(* IEC 61131-3 sources: brOscatLib/oscatNetw, 129 files *)

(* ---- oscatNetw.typ ---- *)
TYPE
    DLOG_CRON_DATA :    STRUCT
        CE : ARRAY[0..5] OF DLOG_CRON_ELEMENT;
    END_STRUCT;
    DLOG_CRON_ELEMENT :    STRUCT
        ELEMENTS : ARRAY[0..59] OF BOOL;
        VALUE : INT;
        VALUE_MIN : INT;
        VALUE_MAX : INT;
        ALL_SELECTED : BOOL;
    END_STRUCT;
    DLOG_DATA :    STRUCT
        STORE_TYPE : BYTE;
        ADD_COM : INT;
        ADD_DATA_REQ : BOOL;
        CLOCK_TRIG : BOOL;
        ID_MAX : USINT;
        DTI : DT;
        UCB : UNI_CIRCULAR_BUFFER_DATA;
        LOAD_TIME_MAX : TIME;
        NEW_FILE : STRING[255];
        NEW_FILE_SIZE : UDINT;
        NEW_FILE_RTRIG : BOOL;
    END_STRUCT;
    DLOG_REAL_ARRAY_ELEMENT :    STRUCT
        VALUE : REAL;
        DELTA : REAL;
        COLUMN : STRING[10];
        _DELTA_LAST : REAL;
        _VALUE_LAST : REAL;
    END_STRUCT;
    DLOG_RETAIN :    STRUCT
        FN_REM : STRING[255];
        COLOR : BOOL;
        HEAD : BOOL;
        TRIG_CNT : UDINT;
        TRIG_CNT_TOTAL : UDINT;
    END_STRUCT;
    DLOG_SAVE :    STRUCT
        FN_REM : STRING[255];
        COLOR : BOOL;
        HEAD : BOOL;
        TRIG_CNT : UDINT;
        TRIG_CNT_TOTAL : UDINT;
    END_STRUCT;
    LOG_CONTROL :    STRUCT
        NEW_MSG : STRING[LOG_SIZE]; (* neue Nachricht für den Datenbuffer *)
        NEW_MSG_OPTION : DWORD;
        LEVEL : BYTE;
        SIZE : INT := LOG_MAX; (* Anzahl der Strings im LOG_DATA *)
        RESET : BOOL; (* Nachrichtenbuffer löschen *)
        PRINTF : PRINTF_DATA; (* Array PRINTF Parameter *)
        MSG : ARRAY[0..LOG_MAX] OF STRING[LOG_SIZE]; (* Array Message *)
        MSG_OPTION : ARRAY[0..LOG_MAX] OF DWORD; (* Array Options *)
        UPDATE_COUNT : UINT; (* Updatezähler *)
        IDX : INT; (* aktueller Nachrichten-Index *)
        RING_MODE : BOOL; (* Bufferüberlauf erkannt *)
    END_STRUCT;
    UNI_CIRCULAR_BUFFER_DATA :    STRUCT
        D_MODE : INT;
        D_SIZE : INT;
        D_HEAD : WORD;
        D_STRING : STRING[STRING_LENGTH];
        D_REAL : REAL;
        D_DWORD : DWORD;
        BUF_SIZE : UINT;
        BUF_COUNT : UINT;
        BUF_USED : USINT;
        BUF_USED_MAX : USINT;
        BUF_DATA_CNT : UDINT;
        BUF_DATA_LOST : UDINT;
        BUF : UNI_CIRCULAR_BUF;
        _GetStart : UINT;
        _GetEnd : UINT;
        _Last : UINT;
        _First : UINT;
    END_STRUCT;
    us_LOG_VIEWPORT :    STRUCT
        LINE_ARRAY : ARRAY[1..40] OF INT;
        COUNT : INT; (* Anzahl der sichtbaren Nachtrichten *)
        UPDATE_COUNT : UINT; (* Updatezähler *)
        MOVE_TO_X : INT; (* Steuerung der Nachrichtenanzeige *)
        UPDATE : BOOL; (* Daten wurden geändert -> neuzeichnen *)
    END_STRUCT;
    MYSQL_COM :    STRUCT
        S_BUF : NETWORK_BUFFER;
        R_BUF : NETWORK_BUFFER;
        SQL_CON : BOOL;
        SQL_URL : STRING[STRING_LENGTH];
        SQL_PACKET_NO : BYTE;
        TIMEOUT : TIME;
        DNS_IP4 : DWORD;
        SQL_RCV_STATE : BYTE;
        ERROR_C : DWORD;
        ERROR_T : BYTE;
    END_STRUCT;
    MYSQL_INFO :    STRUCT
        SERVER_PROTOCOL_VERSION : BYTE;
        SERVER_CAPABILITIES : WORD;
        SERVER_STATUS : WORD;
        SERVER_LANGUAGE : BYTE;
        SQL_CONNECTED : BOOL;
        SQL_ERROR : STRING[STRING_LENGTH];
        DATA_INSERT_AKTIV : BOOL;
        DATA_INSERT_OK_CNT : UDINT;
        DATA_INSERT_NOK_CNT : UDINT;
    END_STRUCT;
    FILE_PATH_DATA :    STRUCT
        DRIVE : STRING[3];
        DIRECTORY : STRING[STRING_LENGTH];
        FILENAME : STRING[255];
    END_STRUCT;
    FILE_SERVER_DATA :    STRUCT
        FILE_OPEN : BOOL;
        FILENAME : STRING[255];
        MODE : BYTE;
        OFFSET : UDINT;
        FILE_SIZE : UDINT;
        ERROR : BYTE;
        RUNTIME : FILE_SERVER_RUNTIME_DATA;
    END_STRUCT;
    FILE_SERVER_RUNTIME_DATA :    STRUCT
        TIME_FILE_OPEN_CUR : UDINT;
        TIME_FILE_OPEN_MAX : UDINT;
        TIME_FILE_OPEN_MIN : UDINT;
        TIME_FILE_CLOSE_CUR : UDINT;
        TIME_FILE_CLOSE_MAX : UDINT;
        TIME_FILE_CLOSE_MIN : UDINT;
        TIME_FILE_READ_CUR : UDINT;
        TIME_FILE_READ_MAX : UDINT;
        TIME_FILE_READ_MIN : UDINT;
        TIME_FILE_WRITE_CUR : UDINT;
        TIME_FILE_WRITE_MAX : UDINT;
        TIME_FILE_WRITE_MIN : UDINT;
        TIME_FILE_SEEK_CUR : UDINT;
        TIME_FILE_SEEK_MAX : UDINT;
        TIME_FILE_SEEK_MIN : UDINT;
        TIME_FILE_TELL_CUR : UDINT;
        TIME_FILE_TELL_MAX : UDINT;
        TIME_FILE_TELL_MIN : UDINT;
        TIME_FILE_DELETE_CUR : UDINT;
        TIME_FILE_DELETE_MAX : UDINT;
        TIME_FILE_DELETE_MIN : UDINT;
    END_STRUCT;
    NET_VAR_DATA :    STRUCT
        CYCLE : UDINT;
        STATE : BYTE;
        INDEX : INT;
        ID_MAX : USINT;
        ERROR_ID : BYTE;
        BUF_SIZE : UINT;
        S_BUF : NETWORK_BUFFER;
        R_BUF : NETWORK_BUFFER;
    END_STRUCT;
    IP2GEO_DATA :    STRUCT
        STATE : BOOL;
        IP4 : DWORD;
        COUNTRY_CODE : STRING[2];
        COUNTRY_NAME : STRING[20];
        REGION_CODE : STRING[2];
        REGION_NAME : STRING[20];
        CITY : STRING[20];
        GEO_LATITUDE : REAL;
        GEO_LONGITUDE : REAL;
        TIME_ZONE_NAME : STRING[20];
        GMT_OFFSET : INT;
        IS_DST : BOOL;
    END_STRUCT;
    IP_C :    STRUCT
        C_MODE : BYTE; (*W Mode: TCP/UCP AKTIV/PASSIV                               *)
        C_PORT : WORD; (*W Portnummer                                               *)
        C_IP : DWORD; (*W IP-Adresse gepackt wwxxyyzz = www.xxx.yyy.zzz            *)
        C_STATE : BYTE; (*R Verbindungsstatus ON/OFF + Flanke ON/OFF                 *)
        C_ENABLE : BOOL; (*W Freigabe für Connect                                     *)
        R_OBSERVE : BOOL; (*W Empfang ueberwachen                                      *)
        TIME_RESET : BOOL; (*W Alle Timer ruecksetzen                                   *)
        ERROR : DWORD; (*R vvwwxxyy (vv = CON_ERROR, ww = SEN_ERROR, xx = REC_ERROR *)
        FIFO : IP_FIFO_DATA; (*I IP FIFO Struktur                                         *)
        MAILBOX : ARRAY[1..16] OF BYTE; (*I Mailbox: Datenbereich für Bausteindatenaustausch         *)
    END_STRUCT;
    IP_FIFO_DATA :    STRUCT
        X : ARRAY[1..128] OF BYTE; (* IP_ID FIFO Speicher          *)
        Y : ARRAY[1..128] OF BYTE; (* IP_ID Zähler                 *)
        ID : BYTE; (* höchste vergabene id         *)
        MAX_ID : BYTE; (* maximal Anmeldungen pro ID   *)
        INIT : BOOL; (* Initialisierung durchgeführt *)
        EMPTY : BOOL; (* FIFO leer                    *)
        FULL : BOOL; (* FIFO voll                    *)
        TOP : INT; (* maximale anzahl in FIFO      *)
        NW : INT; (* Schreibzeiger                *)
        NR : INT; (* Lesezeiger                   *)
    END_STRUCT;
    NETWORK_BUFFER :    STRUCT
        SIZE : UINT;
        BUFFER : NW_BUF_LONG;
    END_STRUCT;
    NETWORK_BUFFER_SHORT :    STRUCT
        SIZE : UINT;
        BUFFER : NW_BUF_SHORT;
    END_STRUCT;
    URL :    STRUCT
        PROTOCOL : STRING[10];
        USER : STRING[32];
        PASSWORD : STRING[32];
        DOMAIN : STRING[80];
        PORT : WORD;
        PATH : STRING[80];
        QUERY : STRING[STRING_LENGTH];
        ANCHOR : STRING[40];
        HEADER : STRING[160];
    END_STRUCT;
    VMAP_DATA :    STRUCT
        FC : DWORD;
        V_ADR : INT;
        V_SIZE : INT;
        P_ADR : INT;
        TIME_OUT : TIME;
    END_STRUCT;
    XML_CONTROL :    STRUCT
        COMMAND : WORD;
        WATCHDOG : TIME;
        START_POS : UINT;
        STOP_POS : UINT;
        COUNT : UINT;
        TYP : INT;
        LEVEL : UINT;
        PATH : STRING[STRING_LENGTH];
        ELEMENT : STRING[STRING_LENGTH];
        ATTRIBUTE : STRING[STRING_LENGTH];
        VALUE : STRING[STRING_LENGTH];
        BLOCK1_START : UINT;
        BLOCK1_STOP : UINT;
        BLOCK2_START : UINT;
        BLOCK2_STOP : UINT;
    END_STRUCT;
    us_TN_INPUT_CONTROL :    STRUCT
        bo_Enable : BOOL; (* Bearbeitung freigeben/sperren *)
        bo_Update_all : BOOL; (* All Elemente neu zeichnen *)
        bo_Reset_Fokus : BOOL; (* Fokus auf 1. Element setzen *)
        in_Focus_at : INT; (* Controlelement mit aktivem Fokus *)
        in_Count : INT; (* Anzahl der benutzen Control-Elemente *)
        in_ToolTip_X : INT; (* Tooltip Text X-Offset *)
        in_ToolTip_Y : INT; (* Tooltip Text Y-Offset *)
        by_ToolTip_Attr : BYTE; (* Tooltip Text Attribute *)
        in_ToolTip_Size : INT; (* Tooltip Text länge *)
        usa_TN_INPUT_CONTROL_DATA : ARRAY[1..20] OF us_TN_INPUT_CONTROL_DATA;
    END_STRUCT;
    us_TN_INPUT_CONTROL_DATA :    STRUCT
        by_Input_Exten_Code : BYTE;
        by_Input_ASCII_Code : BYTE;
        bo_Input_ASCII_IsNum : BOOL;
        in_Title_X_Offset : INT; (* Title Text X-Offset *)
        in_Title_Y_Offset : INT; (* Title Text Y-Offset *)
        by_Title_Attr : BYTE; (* Title Text Attribute *)
        st_Title_String : STRING[255]; (* Title Text String *)
        in_Cursor_X : INT; (* aktuelle Cursor X-Position *)
        in_Cursor_Y : INT; (* aktuelle Cursor Y-Position *)
        in_Type : INT; (* Type des Elements *)
        in_X : INT; (* Element X-Position *)
        in_Y : INT; (* Element Y-Position *)
        in_Cursor_Pos : INT; (* aktuelle Cursorposition *)
        by_Attr_mF : BYTE; (* Text Attribute mit Fokus *)
        by_Attr_oF : BYTE; (* Text Attribute ohne Fokus *)
        in_selected : INT; (* Text Item wurde ausgewählt *)
        st_Input_Mask : STRING[255]; (* Text Eingabemaske *)
        st_Input_Data : STRING[STRING_LENGTH]; (* Text aktuelle Eingabedaten *)
        st_Input_String : STRING[255]; (* Text Kopie nach Return-Taste *)
        st_Input_ToolTip : STRING[255]; (* Text ToolTip (Eingabeinformation) *)
        in_Input_Option : INT; (* Text Ausgabe-Optionen *)
        bo_Input_Entered : BOOL; (* RETURN-Taste wurde betätigt *)
        bo_Input_Hidden : BOOL; (* Text versteckete Eingabe mit '*' *)
        bo_Input_Only_Num : BOOL; (* Text nur Nummerneingabe zulassen *)
        bo_Focus : BOOL; (* Element besitzt den Fokus *)
        bo_Update_Input : BOOL; (* Element wegen Benutzereingabe neuzeichnen *)
        bo_Update_All : BOOL; (* Element komplett neuzeichnen *)
    END_STRUCT;
    us_TN_MENU :    STRUCT
        st_Menu_Text : STRING[STRING_LENGTH]; (* X Menue Texte *)
        in_Menu_E_Count : INT; (* Menue Elemente Anzahl *)
        in_Y : INT; (* Menue Zeilennummer  Y-Position *)
        in_X : INT; (* Menue Spaltennummer X-Position *)
        by_Attr_mF : BYTE; (* Text Attribute mit Fokus *)
        by_Attr_oF : BYTE; (* Text Attribute ohne Fokus *)
        in_X_SM_new : INT; (* neue Sub-Menu X-Position *)
        in_Y_SM_new : INT; (* neue Sub-Menu Y-Position *)
        in_X_SM_old : INT; (* alte Sub-Menu X-Position *)
        in_Y_SM_old : INT; (* alte Sub-Menu Y-Position *)
        in_Cur_Menu_Item : INT; (* aktuelles Haupt-Menue *)
        in_Cur_Sub_Item : INT; (* aktuelles Sub-Menue *)
        in_State : INT; (*   Menu status   *)
        in_Menu_Selected : INT; (* X Menu-Item mit Enter angewwählt *)
        bo_Create : BOOL; (* X Menu erzeugen *)
        bo_Destroy : BOOL; (* X Menu entfernen *)
        bo_Update : BOOL; (* X Menu updaten *)
    END_STRUCT;
    us_TN_MENU_POPUP :    STRUCT
        st_Menu_Text : STRING[STRING_LENGTH]; (* X Menue Texte *)
        in_Menu_E_Count : INT; (* Menue Elemente Anzahl *)
        in_X : INT; (* X Menue X-Position *)
        in_Y : INT; (* X Menue Y-Position *)
        in_Cols : INT; (* Menue Spaltenanzahl *)
        in_Rows : INT; (* Menue Zeilenanzahl *)
        in_Cur_Item : INT; (* X aktuelles Sub-Menue *)
        by_Attr_mF : BYTE; (* X Text Attribute mit Fokus	*)
        by_Attr_oF : BYTE; (* X Text Attribute ohne Fokus *)
        by_Input_Exten_Code : BYTE; (* X Tastencode: Sondertasten *)
        bo_Create : BOOL; (* X Popup-Menu erzeugen *)
        bo_Destroy : BOOL; (* X Popup-Menu entfernen *)
        bo_Update : BOOL; (* X Popup-Menu updaten *)
        bo_Activ : BOOL; (*   Popup-Menu ist aktiv *)
    END_STRUCT;
    us_TN_SCREEN :    STRUCT
        bya_CHAR : ARRAY[0..1919] OF BYTE;
        bya_COLOR : ARRAY[0..1919] OF BYTE;
        bya_BACKUP : ARRAY[0..1919] OF BYTE;
        bya_Line_Update : ARRAY[0..23] OF BOOL;
        by_Input_Exten_Code : BYTE;
        by_Input_ASCII_Code : BYTE;
        bo_Input_ASCII_IsNum : BOOL;
        in_Page_Number : INT; (* aktive Seiten-Nr. *)
        in_Cursor_X : INT; (* Cursor X-Position *)
        in_Cursor_Y : INT; (* Cursor Y-Position *)
        in_EOS_Offset : INT; (* End of String Offset *)
        by_Clear_Screen_Attr : BYTE; (* Clear-Screen Attr *)
        bo_Clear_Screen : BOOL; (* Clear-Screen auslösen *)
        bo_Modal_Dialog : BOOL; (* Modaler Dialog ist aktiv *)
        bo_Menue_Bar_Dialog : BOOL; (* Menue Dialog ist aktiv *)
    END_STRUCT;
    WORLD_WEATHER_CUR :    STRUCT
        OBSERVATION_TIME : STRING[8];
        TEMP_C : INT;
        WEATHER_CODE : INT;
        WEATHER_DESC : STRING[60];
        WEATHER_ICON : INT;
        WIND_SPEED_MILES : INT;
        WIND_SPEED_KMPH : INT;
        WIND_DIR_DEGREE : INT;
        WIND_DIR16POINT : STRING[3];
        PRECIPMM : REAL;
        HUMIDITY : INT;
        VISIBILITY : INT;
        PRESSURE : INT;
        CLOUDOVER : INT;
    END_STRUCT;
    WORLD_WEATHER_DATA :    STRUCT
        CUR : WORLD_WEATHER_CUR;
        DAY : ARRAY[0..4] OF WORLD_WEATHER_DAY;
    END_STRUCT;
    WORLD_WEATHER_DAY :    STRUCT
        DATE_OF_DAY : STRING[10];
        TEMP_MAX_C : INT;
        TEMP_MAX_F : INT;
        TEMP_MIN_C : INT;
        TEMP_MIN_F : INT;
        WIND_SPEED_MILES : INT;
        WIND_SPEED_KMPH : INT;
        WIND_DIR_DEGREE : INT;
        WIND_DIR16POINT : STRING[3];
        WEATHER_CODE : INT;
        WEATHER_DESC : STRING[60];
        WEATHER_ICON : INT;
        PRECIPMM : REAL;
    END_STRUCT;
    YAHOO_WEATHER_DATA :    STRUCT
        LOCATION_CITY : STRING[40]; (* THE LOCATION OF THIS FORECAST: CITY: CITY NAME  *)
        LOCATION_REGION : STRING[20]; (* THE LOCATION OF THIS FORECAST: REGION: STATE, TERRITORY, OR REGION, IF GIVEN *)
        LOCATION_COUNTRY : STRING[20]; (* THE LOCATION OF THIS FORECAST: COUNTRY: TWO-CHARACTER COUNTRY CODE *)
        UNIT_TEMPERATURE : STRING[1]; (* TEMPERATURE: DEGREE UNITS, F FOR FAHRENHEIT OR C FOR CELSIUS *)
        UNIT_DISTANCE : STRING[2]; (* DISTANCE: UNITS FOR DISTANCE, MI FOR MILES OR KM FOR KILOMETERS *)
        UNIT_PRESSURE : STRING[2]; (* PRESSURE: UNITS OF BAROMETRIC PRESSURE, IN FOR POUNDS PER SQUARE INCH OR MB FOR MILLIBARS *)
        UNIT_SPEED : STRING[4]; (* SPEED: UNITS OF SPEED, MPH FOR MILES PER HOUR OR KPH FOR KILOMETERS PER HOUR *)
        WIND_CHILL : INT; (* FORECAST INFORMATION ABOUT WIND CHILL IN DEGREES *)
        WIND_DIRECTION : INT; (* FORECAST INFORMATION ABOUT WIND DIRECTION, IN DEGREES *)
        WIND_SPEED : REAL; (* FORECAST INFORMATION ABOUT WIND SPEED, IN THE UNITS (MPH OR KPH)*)
        ATMOSPHERE_HUMIDITY : INT; (* FORECAST INFORMATION ABOUT CURRENT ATMOSPHERIC HUMIDITY: HUMIDITY, IN PERCENT  *)
        ATMOSPHERE_PRESSURE : REAL; (* FORECAST INFORMATION ABOUT CURRENT ATMOSPHERIC PRESSURE: BAROMETRIC PRESSURE, IN THE UNITS (IN OR MB) *)
        ATMOSPHERE_VISIBILITY : REAL; (* FORECAST INFORMATION ABOUT CURRENT ATMOSPHERIC VISIBILITY, IN THE UNITS (MI OR KM) *)
        ATMOSPHERE_RISING : INT; (* FORECAST INFORMATION ABOUT RISING: STATE OF THE BAROMETRIC PRESSURE: STEADY (0), RISING (1), OR FALLING (2). (INTEGER: 0, 1, 2) *)
        ASTRONOMY_SUNRISE : STRING[10]; (* SUNRISE: TODAY'S SUNRISE TIME. THE TIME IS A STRING IN A LOCAL TIME FORMAT OF "H:MM AM/PM" *)
        ASTRONOMY_SUNSET : STRING[10]; (* SUNSET: TODAY'S SUNSET TIME. THE TIME IS A STRING IN A LOCAL TIME FORMAT OF "H:MM AM/PM", *)
        GEO_LATITUDE : REAL; (* THE LATITUDE OF THE LOCATION *)
        GEO_LONGITUDE : REAL; (* THE LONGITUDE OF THE LOCATION *)
        CUR_CONDITIONS_TEMP : INT; (* THE CURRENT WEATHER CONDITIONS: TEMP: THE CURRENT TEMPERATURE, IN THE UNITS (F OR C) *)
        CUR_CONDITIONS_TEXT : STRING[40]; (* THE CURRENT WEATHER CONDITIONS: TEXT: A TEXTUAL DESCRIPTION OF CONDITIONS *)
        CUR_CONDITIONS_CODE : INT; (* THE CURRENT WEATHER CONDITIONS: CODE: THE CONDITION CODE FOR THIS FORECAST *)
        CUR_CONDITIONS_ICON : INT; (* THE CURRENT WEATHER CONDITIONS: ICON: THE CONDITION ICON FOR THIS FORECAST *)
        FORECAST_TODAY_LOW_TEMP : INT; (* THE FORECAST TODAY WEATHER CONDITIONS: THE FORECASTED LOW TEMPERATURE FOR THIS DAY IN THE UNITS (F OR C) *)
        FORECAST_TODAY_HIGH_TEMP : INT; (* THE FORECAST TODAY WEATHER CONDITIONS: THE FORECASTED HIGH TEMPERATURE FOR THIS DAY IN THE UNITS (F OR C) *)
        FORECAST_TODAY_TEXT : STRING[40]; (* THE FORECAST TODAY WEATHER CONDITIONS: TEXT: A TEXTUAL DESCRIPTION OF CONDITIONS *)
        FORECAST_TODAY_CODE : INT; (* THE CURRENT WEATHER CONDITIONS: CODE: THE CONDITION CODE FOR THIS FORECAST *)
        FORECAST_TODAY_ICON : INT; (* THE CURRENT WEATHER CONDITIONS: ICON: THE CONDITION ICON FOR THIS FORECAST *)
        FORECAST_TODAY_DATE_LONG : STRING[20]; (* THE CURRENT WEATHER CONDITIONS: DATE: DATE OF THE DAY *)
        FORECAST_DAY : ARRAY[1..9] OF YAHOO_WEATHER_FORECAST_DAY; (* THE CURRENT WEATHER DAYS ARRAY *)
    END_STRUCT;
    YAHOO_WEATHER_FORECAST_DAY :    STRUCT
        LOW_TEMP : INT; (* THE FORECAST WEATHER CONDITIONS: THE FORECASTED LOW TEMPERATURE FOR THIS DAY IN THE UNITS (F OR C) *)
        HIGH_TEMP : INT; (* THE FORECAST WEATHER CONDITIONS: THE FORECASTED HIGH TEMPERATURE FOR THIS DAY IN THE UNITS (F OR C) *)
        TEXT : STRING[40]; (* THE FORECAST WEATHER CONDITIONS: TEXT: A TEXTUAL DESCRIPTION OF CONDITIONS *)
        DATE_LONG : STRING[20]; (* THE FORECAST WEATHER CONDITIONS: DATE: DATE OF THE DAY *)
        CODE : INT; (* THE FORECAST WEATHER CONDITIONS: CODE: THE CONDITION CODE FOR THIS FORECAST *)
        ICON : INT; (* THE FORECAST WEATHER CONDITIONS: ICON: THE CONDITION ICON FOR THIS FORECAST *)
    END_STRUCT;
END_TYPE

(* ---- ELEMENT_COUNT.st ---- *)
FUNCTION ELEMENT_COUNT
    (*http://www.oscat.de/images/OSCATNetwork/oscat_netlib121_en.pdf#page=34*)
    IF ELEMENT = '' THEN
    	ELEMENT_COUNT := 0;
    ELSE
    	pt := ADR(ELEMENT);
    	ELEMENT_COUNT := 1;
    	l := LEN(ELEMENT);
    	FOR pos := 1 TO l DO
    		IF pt[pos] = SEP THEN ELEMENT_COUNT := ELEMENT_COUNT + 1; END_IF
    	END_FOR
    END_IF

    (* revision histroy
    ks	5. apr. 2011	rev 1.0
    	original release

    *)
END_FUNCTION

(* ---- ELEMENT_GET.st ---- *)
FUNCTION ELEMENT_GET
    (*http://www.oscat.de/images/OSCATNetwork/oscat_netlib121_en.pdf#page=34*)
    (* load pointers *)
    pt := ADR(ELEMENT);
    po := ADR(ELEMENT_GET);

    (* search for the n-th occurence of a separation character and store position in i *)
    WHILE (cnt < POS) AND (i < ELEMENT_LENGTH) AND (pt[i] > 0) DO
    	IF pt[i] = SEP THEN cnt := cnt + 1; END_IF
    	i := i + 1;
    END_WHILE

    (* copy the list ELEMENT to output *)
    IF i < ELEMENT_LENGTH THEN c := pt[i]; END_IF
    WHILE (c <> SEP) AND (c > 0) AND (o < ELEMENT_LENGTH) AND (i < ELEMENT_LENGTH) DO
    	po[o] :=pt[i];
    	o := o + 1;
    	i := i + 1;
    	c := pt[i];
    END_WHILE

    (* terminate the output string *)
    po[o] := 0;

    (* revision histroy
    ks 05. apr. 2011	rev 1.0
    	original release

    *)
END_FUNCTION

(* ---- FILE_PATH_SPLIT.st ---- *)
FUNCTION FILE_PATH_SPLIT
    (*http://www.oscat.de/images/OSCATNetwork/oscat_netlib121_en.pdf#page=153*)
    X.DRIVE := '';
    X.DIRECTORY := '';
    X.FILENAME := '';
    c := LEN(FILENAME);
    IF c = 0 THEN
    	FILE_PATH_SPLIT := FALSE;
    	RETURN;
    END_IF

    FOR b := 1 TO c DO
    	d := MID(FILENAME, 1, b);
    	IF d = ':' THEN
    		p1 := b;
    	ELSIF d = '/' OR d = '\' THEN
    		p2 := b;
    	END_IF
    END_FOR

    IF p1 = 2 THEN
    	X.DRIVE := LEFT(FILENAME,p1);
    END_IF

    IF p2 > 0 AND p2 > p1 THEN
    	X.DIRECTORY := MID(FILENAME,p2 - p1,p1+1); (* len , pos *)
    END_IF

    X.FILENAME := RIGHT(FILENAME,c - MAX (p1,p2));
    FILE_PATH_SPLIT := TRUE;

    (* revision history
    ks	01. jan. 2011	rev 1.0
    	original version
    *)
END_FUNCTION

(* ---- HTML_DECODE.st ---- *)
FUNCTION HTML_DECODE
    (*http://www.oscat.de/images/OSCATNetwork/oscat_netlib121_en.pdf#page=75*)
    HTML_DECODE := IN;

    (* docode characters encoded by character position *)
    pos := FIND(HTML_DECODE, '&');
    WHILE pos > 0 DO
    	tmp := MID(HTML_DECODE, 2, pos + 1);
    	IF tmp = '#x' OR tmp = '#X' THEN
    		(* hexadecimal representation found *)
    		tmp := MID(HTML_DECODE, 10, pos + 3);
    		end := FIND(tmp, ';');
    		code := CHR_TO_STRING(DWORD_TO_BYTE(HEX_TO_DWORD(LEFT(tmp, end - 1))));
    		HTML_DECODE := REPLACE(HTML_DECODE, code, end + 3, pos);
    	ELSIF LEFT(tmp,1) = '#' THEN
    		tmp := MID(HTML_DECODE, 10, pos + 2);
    		end := FIND(tmp, ';');
    		code := CHR_TO_STRING(INT_TO_BYTE(STRING_TO_INT(LEFT(tmp, end - 1))));
    		HTML_DECODE := REPLACE(HTML_DECODE, code, end + 2, pos);
    	ELSE
    		(* replace all named characters *)
    		tmp := MID(HTML_DECODE, 10, pos + 1);
    		end := FIND(tmp, ';');
    		code := CHR_TO_STRING(CHARCODE(LEFT(tmp, end - 1)));
    		HTML_DECODE := REPLACE(HTML_DECODE, code, end + 1, pos);
    	END_IF
    	(* search for next occurence of encoded characters *)
    	pos := FINDP(HTML_DECODE, '&', pos + 1);
    END_WHILE

    (* revision history
    hm	3. mai. 2008	rev 1.0
    	original version

    hm	16. jun. 2008	rev 1.1
    	changed nested call of replace for better compatibility

    hm	17. dec. 2008	rev 1.2
    	changed function CHR to CHR_TO_STRING

    hm	10. may. 2010	rev 1.3
    	stringlength 250

    *)
END_FUNCTION

(* ---- HTML_ENCODE.st ---- *)
FUNCTION HTML_ENCODE
    (*http://www.oscat.de/images/OSCATNetwork/oscat_netlib121_en.pdf#page=76*)
    pt_in  := ADR(IN);
    pt_out := ADR(HTML_ENCODE);

    (* scan the input string and convert unallowed characters *)
    pos_in := 1;
    stop := LEN(IN);
    FOR pos_out := 1 TO 250 DO
    	IF pos_in > stop THEN EXIT; END_IF
    	B := pt_in[pos_in];
    	CASE BYTE_TO_INT(B) OF
    		34: (* " detected *)
    			IF pos_out > STRING_LENGTH - 6 THEN EXIT; END_IF
    			pt_out[pos_out] := 38;
    			pos_out := pos_out + 1;
    			pt_out[pos_out] := 113;
    			pos_out := pos_out + 1;
    			pt_out[pos_out] := 117;
    			pos_out := pos_out + 1;
    			pt_out[pos_out] := 111;
    			pos_out := pos_out + 1;
    			pt_out[pos_out] := 116;
    			pos_out := pos_out + 1;
    			pt_out[pos_out] := 59;
    		38: (* & detected *)
    			IF pos_out > STRING_LENGTH - 5 THEN EXIT; END_IF
    			pt_out[pos_out] := 38;
    			pos_out := pos_out + 1;
    			pt_out[pos_out] := 97;
    			pos_out := pos_out + 1;
    			pt_out[pos_out] := 109;
    			pos_out := pos_out + 1;
    			pt_out[pos_out] := 112;
    			pos_out := pos_out + 1;
    			pt_out[pos_out] := 59;
    		60: (* < detected *)
    			IF pos_out > STRING_LENGTH - 4 THEN EXIT; END_IF
    			pt_out[pos_out] := 38;
    			pos_out := pos_out + 1;
    			pt_out[pos_out] := 108;
    			pos_out := pos_out + 1;
    			pt_out[pos_out] := 116;
    			pos_out := pos_out + 1;
    			pt_out[pos_out] := 59;
    		62: (* > detected *)
    			IF pos_out > STRING_LENGTH - 4 THEN EXIT; END_IF
    			pt_out[pos_out] := 38;
    			pos_out := pos_out + 1;
    			pt_out[pos_out] := 103;
    			pos_out := pos_out + 1;
    			pt_out[pos_out] := 116;
    			pos_out := pos_out + 1;
    			pt_out[pos_out] := 59;
    	ELSE
    		IF M AND B > 127 THEN
    			tmp := CHARNAME(B);
    			(* exit if output string has not enough space *)
    			IF pos_out + LEN(tmp) + 2 <= 250 THEN
    				pt_out[pos_out] := 38;
    				pos_out := pos_out + 1;
    				FOR i := 1 TO LEN(tmp) DO
    					pt_out[pos_out] := CODE(tmp, i);
    					pos_out := pos_out + 1;
    				END_FOR
    				pt_out[pos_out] := 59;
    			END_IF
    		ELSE
    			pt_out[pos_out] := B;
    		END_IF
    	END_CASE
    	(* increment IN by 1 *)
    	pos_in := pos_in + 1;
    END_FOR

    (* terminate the output string *)
    pt_out[pos_out] := 0;

    (* revision history
    hm		3. mai. 2008	rev 1.0
    	original version

    hm		10. mai. 2008	rev 1.1
    	stringlength 250
    *)
END_FUNCTION

(* ---- IP4_CHECK.st ---- *)
FUNCTION IP4_CHECK
    (*http://www.oscat.de/images/OSCATNetwork/oscat_netlib121_en.pdf#page=77*)
    IP4_CHECK := (NIP AND SM) = (LIP AND SM);

    (* revision history
    hm		4. mar 2008	rev 1.0
    	original version

    *)
END_FUNCTION

(* ---- IP4_DECODE.st ---- *)
FUNCTION IP4_DECODE
    (*http://www.oscat.de/images/OSCATNetwork/oscat_netlib121_en.pdf#page=77*)
    pos := FIND(STR, '.');
    WHILE pos > 0 DO
    	IP4_DECODE := SHL(IP4_DECODE,8) OR STRING_TO_DWORD(LEFT(STR,pos - 1));
    	STR := DELETE(STR, pos, 1);
    	pos := FIND(STR, '.');
    END_WHILE
    IP4_DECODE := SHL(IP4_DECODE,8) OR STRING_TO_DWORD(STR);

    (* revision history
    hm		29. feb 2008	rev 1.0
    	original version

    hm	10. mar. 2009	rev 1.1
    	new algorythm
    *)
END_FUNCTION

(* ---- IP4_TO_STRING.st ---- *)
FUNCTION IP4_TO_STRING
    (*http://www.oscat.de/images/OSCATNetwork/oscat_netlib121_en.pdf#page=78*)
    (* mask bits AND INSERT AT given position *)
    tmp := BYTE_TO_STRING(DWORD_TO_BYTE(IP4));
    IP4_TO_STRING := CONCAT('...', tmp);
    tmp := BYTE_TO_STRING(DWORD_TO_BYTE(SHR(IP4,8)));
    IP4_TO_STRING := INSERT(IP4_TO_STRING, tmp, 2);
    tmp := BYTE_TO_STRING(DWORD_TO_BYTE(SHR(IP4,16)));
    IP4_TO_STRING := INSERT(IP4_TO_STRING, tmp, 1);
    tmp := BYTE_TO_STRING(DWORD_TO_BYTE(SHR(IP4,24)));
    IP4_TO_STRING := CONCAT(tmp, IP4_TO_STRING);

    (* revision history
    hm	22. apr 2008	rev 1.0
    	original version

    hm	10. mar. 2009	rev 1.1
    	improved code
    *)
END_FUNCTION

(* ---- IS_IP4.st ---- *)
FUNCTION IS_IP4
    (*http://www.oscat.de/images/OSCATNetwork/oscat_netlib121_en.pdf#page=78*)
    IS_IP4 := COUNT_CHAR(STR, 46) = 3;

    (* revision history
    hm	1. mar. 2008	rev 1.0
    	original version

    hm	10. mar. 2009	rev 1.1
    	new code

    *)
END_FUNCTION

(* ---- IS_URLCHR.st ---- *)
FUNCTION IS_URLCHR
    (*http://www.oscat.de/images/OSCATNetwork/oscat_netlib121_en.pdf#page=79*)
    IS_URLCHR := ((IN > 47) AND (IN < 58)) OR ((IN > 64) AND (IN < 91)) OR ((IN > 96) AND (IN < 123)) OR (IN = 126) OR (IN = 95) OR (IN =45) OR (IN =46);

    (* revision history
    hm		27. apr. 2008	rev 1.0
    	original version

    *)
END_FUNCTION

(* ---- MD5_AUX.st ---- *)
FUNCTION MD5_AUX
    (*http://www.oscat.de/images/OSCATNetwork/oscat_netlib121_en.pdf#page=79*)
    CASE N OF
    	1: w := (B AND C) OR (NOT(B) AND D);
    	2: w := (B AND D) OR (C AND NOT D);
    	3: w := (B XOR C XOR D);
    	4: w := (C XOR (B OR  NOT(D)));
    END_CASE

    MD5_AUX := B + ROL(A + w + X + T,U);

    (* revision history

    ks	6. dec. 2009 rev 1.0
    	original version

    *)
END_FUNCTION

(* ---- MD5_TO_STRH.st ---- *)
FUNCTION MD5_TO_STRH
    (*http://www.oscat.de/images/OSCATNetwork/oscat_netlib121_en.pdf#page=82*)
    pt := ADR(MD5_TO_STRH); (* read output adress to pointer *)

    FOR i := 0 TO 15 DO; (* write the 8 hex characters backwards *)
    	tmp := SHR(MD5[i],4);
    	pt := tmp + SEL(tmp <= 9,87,48);
    	pt := pt + 1; (* decrement the pointer *)
    	tmp := MD5[i] AND 2#1111;
    	pt := tmp + SEL(tmp <= 9,87,48);
    	pt := pt + 1; (* decrement the pointer *)
    END_FOR
    pt:= 0; (* write the closing byte for the string *)

    (* revision history

    ks	6. dec. 2009 rev 1.0
    	original version

    *)
END_FUNCTION

(* ---- NETWORK_VERSION.st ---- *)
FUNCTION NETWORK_VERSION
    (*http://www.oscat.de/images/OSCATNetwork/oscat_netlib121_en.pdf#page=35*)
    IF IN THEN
    	NETWORK_VERSION := DATE_TO_DWORD(D#2016-07-01);
    ELSE
    	NETWORK_VERSION := 135;
    END_IF

    (* revision history
    ks	2. feb 2011	rev 1.0
    	original version

    *)
END_FUNCTION

(* ---- SHA1_TO_STRH.st ---- *)
FUNCTION SHA1_TO_STRH
    (*http://www.oscat.de/images/OSCATNetwork/oscat_netlib121_en.pdf#page=85*)
    pt := ADR(SHA1_TO_STRH); (* read output adress to pointer *)

    FOR i := 0 TO 19 DO; (* write the 10 hex characters backwards *)
    	tmp := SHR(SHA1[i],4);
    	pt := tmp + SEL(tmp <= 9,87,48);
    	pt := pt + 1; (* decrement the pointer *)
    	tmp := SHA1[i] AND 2#1111;
    	pt := tmp + SEL(tmp <= 9,87,48);
    	pt := pt + 1; (* decrement the pointer *)
    END_FOR
    pt:= 0; (* write the closing byte for the string *)

    (* revision history

    ks	6. dec. 2009 rev 1.0
    	original version

    ks	3. dec. 2011 rev 1.1
    	incorrect string size
    *)
END_FUNCTION

(* ---- STRING_TO_URL.st ---- *)
FUNCTION STRING_TO_URL
    (*http://www.oscat.de/images/OSCATNetwork/oscat_netlib121_en.pdf#page=86*)
    (*

    http://hans:geheim@www.example.org:80/demo/example.cgi?land=de&stadt=aa#abschnitt1
    |       |      |         |         |   |                   |               |
    |       |      |         Host      |   Pfad                Query           Anker
    |       |      Passwort            Port
    |       Benutzer
    Protokoll

    *)

    (* check if string is empty and return empty url *)
    IF STR = '' THEN RETURN; END_IF

    (* extract the protocol *)
    (* first we check if the optional protocol is specified ending with a :// *)
    pos := FIND(STR, '://');
    IF pos > 0 THEN
    	(* store protocol and restore the rest of url in temp *)
    	STRING_TO_URL.PROTOCOL := LEFT(STR, pos - 1);
    	x := RIGHT(STR, LEN(STR) - pos - 2);
    ELSE
    	x := STR;
    	STRING_TO_URL.PROTOCOL := DEFAULT_PROTOCOL;
    END_IF

    (* extract user and password if present ending with a @ *)
    pos := FINDB(STR1:=x,STR2:='@'); (* Find last @ *)

    IF pos > 0 THEN
    	(* extract user *)
    	pos2 := FIND(x,':')+1;
    	IF pos2 > 1 AND pos2 <= pos THEN
    		STRING_TO_URL.USER := LEFT(x,pos2 - 2);
    		STRING_TO_URL.PASSWORD := MID(x, pos - pos2, pos2);
    	ELSE
    		STRING_TO_URL.USER := LEFT(x, pos - 2);
    		STRING_TO_URL.PASSWORD := '';
    	END_IF
    	x := RIGHT(x, LEN(x) - pos);
    ELSE
    	STRING_TO_URL.USER := '';
    	STRING_TO_URL.PASSWORD := '';
    END_IF

    (* extract anchor *)
    pos := FIND(x, '#');
    IF pos > 0 THEN
    	STRING_TO_URL.ANCHOR := RIGHT(x, LEN(x) - pos);
    	x := LEFT(x, pos - 1);
    ELSE
    	STRING_TO_URL.ANCHOR := '';
    END_IF

    (* extract query  *)
    pos := FIND(x, '?');
    IF pos > 0 THEN
    	STRING_TO_URL.QUERY := RIGHT(x, LEN(x) - pos);
    	x := LEFT(x, pos - 1);
    ELSE
    	STRING_TO_URL.QUERY := '';
    END_IF

    (* extract path  *)
    pos := FIND(x, '/');
    IF pos > 0 THEN
    	STRING_TO_URL.PATH := RIGHT(x, LEN(x) - pos + 1);
    	x := LEFT(x, pos - 1);
    ELSE
    	STRING_TO_URL.PATH := DEFAULT_PATH;
    END_IF

    (* extract port and leave domain *)
    pos := FIND(x, ':');
    IF pos > 0 THEN
    	STRING_TO_URL.PORT := STRING_TO_WORD(RIGHT(x, LEN(x) - pos));
    	STRING_TO_URL.DOMAIN := LEFT(x, pos - 1);
    ELSE
    	STRING_TO_URL.PORT := 0;
    	STRING_TO_URL.DOMAIN := x;
    END_IF

    (* revision history
    hm		18. apr 2008	rev 1.0
    	original version

    ks		20. dec. 2010	rev 1.1
    	stringlength 250 , var x

    ks		27. oct. 2012	rev 1.2
    	var_temp zu var geändert

    ks		04. mar. 2016	rev 1.3
    	@ zeichen wird nun von rechts nach links gesucht
    	ermöglicht username und password mit @ zeichen
    *)
END_FUNCTION

(* ---- TN_SC_SHADOW_ATTR.st ---- *)
FUNCTION TN_SC_SHADOW_ATTR
    (*http://www.oscat.de/images/OSCATNetwork/oscat_netlib121_en.pdf#page=191*)
    (* Background Farbe auf Schwarz ändern      *)
    (* und dunkle Fordergrundfarben einschalten *)
    TN_SC_SHADOW_ATTR := ((IBY_ATTR AND BYTE#2#11110000) OR BYTE#2#00001000);

    (* revision history
    ks	10. mai. 2010	rev 1.0
    	original version
    *)
END_FUNCTION

(* ---- TN_SC_XY2_ERROR.st ---- *)
FUNCTION TN_SC_XY2_ERROR
    (*http://www.oscat.de/images/OSCATNetwork/oscat_netlib121_en.pdf#page=196*)
    (* min und max werte prüfen *)
    TN_SC_XY2_ERROR := Y1 < 0 OR X1 < 0 OR Y2 < 0 OR X2 < 0 OR Y1 > 23 OR X1 > 79 OR Y2 > 23 OR X2 > 79;

    (* revision history
    ks	10. mai. 2010	rev 1.0
    	original version
    *)
END_FUNCTION

(* ---- TN_SC_XY_ERROR.st ---- *)
FUNCTION TN_SC_XY_ERROR
    (*http://www.oscat.de/images/OSCATNetwork/oscat_netlib121_en.pdf#page=195*)
    (* min und max werte prüfen *)
    TN_SC_XY_ERROR := Y < 0 OR X < 0 OR Y > 23 OR X > 79;

    (* revision history
    ks	10. mai. 2010	rev 1.0
    	original version
    *)
END_FUNCTION

(* ---- URL_DECODE.st ---- *)
FUNCTION URL_DECODE
    (*http://www.oscat.de/images/OSCATNetwork/oscat_netlib121_en.pdf#page=87*)
    URL_DECODE := IN;
    pos := FIND(URL_DECODE,'%');
    WHILE pos > 0 DO
    	seq := MID(URL_DECODE,2,pos + 1);
    	new := CHR_TO_STRING(DWORD_TO_BYTE(HEX_TO_DWORD(seq)));
    	URL_DECODE := REPLACE(URL_DECODE, new, 3, pos);
    	pos := FIND(URL_DECODE,'%');
    END_WHILE

    (* revision history
    hm	27. apr. 2008	rev 1.0
    	original version

    hm	17. dec. 2008	rev 1.1
    	changes name of function chr to chr_to_string

    ks	10. mai. 2008	rev 1.2
    	stringlength 250
    *)
END_FUNCTION

(* ---- URL_ENCODE.st ---- *)
FUNCTION URL_ENCODE
    (*http://www.oscat.de/images/OSCATNetwork/oscat_netlib121_en.pdf#page=87*)
    pt_in  := ADR(IN);
    pt_out := ADR(URL_ENCODE);

    (* scan the input string and convert unallowed characters *)
    pos_in := 1;
    stop := LEN(IN);
    FOR pos_out := 1 TO 250 DO
    	IF pos_in > stop THEN
    		EXIT;
    	ELSIF IS_URLCHR(pt_in[pos_in]) THEN
    		pt_out[pos_out] := pt_in[pos_in];
    		(* increment IN by 1 *)
    		pos_in := pos_in + 1;
    	ELSE
    		(* cannot fit 3 digits, exit *)
    		IF pos_out > 248 THEN EXIT; END_IF
    		(* invalid character that needs to be converted *)
    		pt_out[pos_out] := 37;    (* start with % sign *)
    		pos_out := pos_out + 1;
    		(* need to add the two hex digits *)
    		tb := SHR(pt_in[pos_in],4);
    		IF tb > 9 THEN
    			pt_out[pos_out] := tb + 55;
    		ELSE
    			pt_out[pos_out] := tb + 48;
    		END_IF
    		pos_out := pos_out + 1;
    		tb := pt_in[pos_in] AND 16#0F;
    		IF tb > 9 THEN
    			pt_out[pos_out] := tb + 55;
    		ELSE
    			pt_out[pos_out] := tb + 48;
    		END_IF
    		(* increment IN and out because out has to move 3 digits *)
    		pos_in := pos_in + 1;
    	END_IF
    END_FOR

    (* terminate the output string *)
    pt_out[pos_out] := 0;

    (* revision history
    hm	27. apr. 2008	rev 1.0
    	original version

    ks	10. mai. 2008	rev 1.1
    	stringlength 250

    *)
END_FUNCTION

(* ---- URL_TO_STRING.st ---- *)
FUNCTION URL_TO_STRING
    (*http://www.oscat.de/images/OSCATNetwork/oscat_netlib121_en.pdf#page=87*)
    (*

    http://hans:geheim@www.example.org:80/demo/example.cgi?land=de&stadt=aa#abschnitt1
    |         |         |                  |                                |   |                                    |                                    |
    |         |         |                 Host                         |   Pfad                            Query                           Anker
    |         |         Passwort                                  Port
    |        Benutzer
    Protokoll

    *)

    (* attach protocol *)
    IF IN.PROTOCOL <> '' THEN URL_TO_STRING := CONCAT(IN.PROTOCOL,'://'); END_IF

    (* attach user and password *)
    IF IN.USER <> '' THEN
    	URL_TO_STRING := CONCAT(URL_TO_STRING, IN.USER);
    	IF IN.PASSWORD <> '' THEN
    		URL_TO_STRING := CONCAT(URL_TO_STRING, ':');
    		URL_TO_STRING := CONCAT(URL_TO_STRING, IN.PASSWORD);
    	END_IF
    	URL_TO_STRING := CONCAT(URL_TO_STRING, '@');
    END_IF

    (* attach domain *)
    URL_TO_STRING := CONCAT(URL_TO_STRING, IN.DOMAIN);

    (* attach Port *)
    IF IN.PORT > 0 THEN
    	URL_TO_STRING := CONCAT(URL_TO_STRING, ':');
    	URL_TO_STRING := CONCAT(URL_TO_STRING, WORD_TO_STRING(IN.PORT));
    END_IF

    (* attach path *)
    URL_TO_STRING := CONCAT(URL_TO_STRING, IN.PATH);

    (* attach query *)
    IF IN.QUERY <> '' THEN
    	URL_TO_STRING := CONCAT(URL_TO_STRING, '?');
    	URL_TO_STRING := CONCAT(URL_TO_STRING, IN.QUERY);
    END_IF

    (* attach anchor *)
    IF IN.ANCHOR <> '' THEN
    	URL_TO_STRING := CONCAT(URL_TO_STRING, '#');
    	URL_TO_STRING := CONCAT(URL_TO_STRING, IN.ANCHOR);
    END_IF

    (* revision history
    hm	18. apr 2008	rev 1.0
    	original version

    ks	10. mai. 2008	rev 1.1
    	stringlength 250
    *)
END_FUNCTION

(* ---- BASE64_DECODE_STR.st ---- *)
FUNCTION_BLOCK BASE64_DECODE_STR
    (*http://www.oscat.de/images/OSCATNetwork/oscat_netlib121_en.pdf#page=72*)
    CASE mode OF
    0:	IF RUN AND NOT run_last THEN
    		DONE := FALSE;
    		mode := 1;
    		end := LEN(STR1);
    		pos := 0;
    		STR2 := '';
    	END_IF
    1:
    	size1 := MIN(48,end - pos);
    	IF size1 > 0 THEN
    		_STRING_TO_BUFFER(STR:=MID(STR1, size1, pos + 1), pos:=0, PT:=ADR(buf1), SIZE:=SIZEOF(buf1));
    		BASE64_DECODE_STREAM(buf1:=buf1 ,buf2:=buf2 ,size1:=size1 ,size2=>size2);
    		STR2 := CONCAT(STR2,BUFFER_TO_STRING(PT:=ADR(buf2), SIZE:=SIZEOF(buf2), START:=0, STOP:=size2 - 1));
    	ELSE
    		mode := 0;
    		DONE := TRUE;
    	END_IF
    	pos := pos + size1;
    END_CASE

    run_last := RUN;

    (* revision history

    ks	6. dec. 2009 rev 1.0
    	original version

    *)
END_FUNCTION_BLOCK

(* ---- BASE64_DECODE_STREAM.st ---- *)
FUNCTION_BLOCK BASE64_DECODE_STREAM
    (*http://www.oscat.de/images/OSCATNetwork/oscat_netlib121_en.pdf#page=73*)
    IF SIZE1 <= 0 THEN SIZE2 := 0; RETURN; END_IF
    c := SIZE1 - 1;
    i2 := 0;
    a := 0;
    b := 0;
    FOR i1 := 0 TO c DO
    	o := BUF1[i1];
    	IF o = 61  (* = *) THEN	EXIT;
    	ELSIF o > 96 (* a-z *) THEN off := 71;
    	ELSIF o > 64 (* a-Z *) THEN off := 65;
    	ELSIF o > 47 (* 0-9 *) THEN off := -4;
    	ELSIF o = 43 (* + *) THEN off := -19;
    	ELSIF o = 47 (* / *) THEN off := -16;
    	END_IF
    	b := SHL(b,6) OR INT_TO_BYTE(o - off);
    	a := a + 6;
    	IF a >= 8 THEN
    		a := a - 8;
    		BUF2[i2] := WORD_TO_BYTE(SHR(b,a));
    		i2 := i2 + 1;
    		b := b AND NOT SHL(WORD#16#FFFF,a);
    	END_IF
    END_FOR
    SIZE2 := i2;

    (* revision history

    ks	6. dec. 2009 rev 1.0
    	original version

    *)
END_FUNCTION_BLOCK

(* ---- BASE64_ENCODE_STR.st ---- *)
FUNCTION_BLOCK BASE64_ENCODE_STR
    (*http://www.oscat.de/images/OSCATNetwork/oscat_netlib121_en.pdf#page=74*)
    CASE mode OF
    0:	IF RUN AND NOT run_last THEN
    		DONE := FALSE;
    		mode := 1;
    		end := LEN(STR1);
    		pos := 0;
    		STR2 := '';
    	END_IF
    1:
    	size1 := MIN(48,end - pos);
    	IF size1 > 0 THEN
    		_STRING_TO_BUFFER(STR:=MID(STR1, size1, pos + 1), pos:=0, PT:=ADR(buf1), SIZE:=SIZEOF(buf1));
    		BASE64_ENCODE_STREAM(buf1:=buf1 ,buf2:=buf2 ,size1:=size1 ,size2=>size2);
    		STR2 := CONCAT(STR2,BUFFER_TO_STRING(PT:=ADR(buf2), SIZE:=SIZEOF(buf2), START:=0, STOP:=size2 - 1));
    	ELSE
    		mode := 0;
    		DONE := TRUE;
    	END_IF
    	pos := pos + size1;
    END_CASE

    run_last := RUN;

    (* revision history

    ks	6. dec. 2009 rev 1.0
    	original version

    *)
END_FUNCTION_BLOCK

(* ---- BASE64_ENCODE_STREAM.st ---- *)
FUNCTION_BLOCK BASE64_ENCODE_STREAM
    (*http://www.oscat.de/images/OSCATNetwork/oscat_netlib121_en.pdf#page=74*)
    IF SIZE1 <= 0 THEN
    	SIZE2 := 0;
    	RETURN;
    END_IF
    c := SIZE1 - 1;
    i2 := 0;
    a := 0;
    b := 0;
    FOR i := 0 TO c DO
    	b := SHL(b,8) OR BUF1[i];
    	a := a + 8;
    	WHILE a >= 6 DO
    		a := a - 6;
    		BUF2[i2] := CODE(BASE64,WORD_TO_INT(SHR(b,a)) + 1);
    		i2 := i2 + 1;
    		b := b AND NOT SHL(WORD#16#FFFF,a);
    	END_WHILE
    END_FOR
    IF a > 0 THEN
    	BUF2[i2] := CODE(BASE64,WORD_TO_INT(SHL(b,6 - a)) + 1);
    	i2 := i2 + 1;
    	i3 := i2 + (NOT INT_TO_WORD(i2) AND 2#11);
    	FOR i := i2 TO i3 DO
    		BUF2[i] := 61;
    	END_FOR
    	SIZE2 := i3 + 1;
    ELSE
    	SIZE2 := i2;
    END_IF

    (* revision history

    ks	6. dec. 2009 rev 1.0
    	original version

    *)
END_FUNCTION_BLOCK

(* ---- CSV_PARSER_BUF.st ---- *)
FUNCTION_BLOCK CSV_PARSER_BUF
    (*http://www.oscat.de/images/OSCATNetwork/oscat_netlib121_en.pdf#page=147*)
    IF RUN > 0 THEN
    	IF state = 0 THEN (* Auswertung neu beginnen *)

    		pv := ADR(VALUE);
    		pv := 0; (* VALUE = '' *)
    		pve := pv + INT_TO_DWORD(STRING_LENGTH);
    		i := UDINT_TO_INT(OFFSET);
    		size := UINT_TO_INT(PT.size) - 1;
    		RESULT := 0;
    		state := 5; (* Befehl in Arbeit (Busy) *)
    		step := 0; (* Auswertung neu beginnen *)

    		(* ---------------- Debug-Message -----------------------*)
    		(*IF _debug_enable THEN
    			LOG_CL.NEW_MSG := 'CPF: Startindex: ~1';
    			LOG_CL.PRINTF[1] := INT_TO_STRING(i);
    			LOG_MSG();
    		END_IF*)
    		(* -----------------------------------------------------------------*)

    	END_IF

    	watchdog(IN:=FALSE,PT:=T#1ms); (* Timer neustarten *)
    	watchdog.IN := TRUE;

    	WHILE (state = 5) DO (* Schleife solange kein Ergebnis *)

    		watchdog(); (* Timer aktualisieren *)

    		IF watchdog.Q THEN (* watchdog ausgelöst *)
    			state := 5;
    			EXIT;
    		ELSIF i > size THEN (* kein weiteres zeichen vorhanden *)
    			state := 10; (* nichts gefunden - Daten-Ende erreicht *)
    			EXIT;
    		ELSE

    			c := PT.BUFFER[i]; (* neues Zeichen aus Buffer lesen *)
    			eof := i + 1 = PT.size; (* End of File *)

    			v_add := 0;

    			IF c = SEP THEN (* Neues Element erkannt *)
    				state := 1;
    				x := TRUE;
    			ELSIF c >= 32 THEN (* Element erkannt *)
    				v_add := c; (* Zeichen ablegen *)
    				IF eof THEN
    					state := 2; (* Element und Zeilenende erkannt *)
    				ELSE
    					x := TRUE;
    				END_IF
    			ELSE
    				IF x THEN
    					state := 2; (* Element und Zeilenende erkannt *)
    					x := FALSE;
    				END_IF
    			END_IF

    			IF v_add > 0  AND pv < pve THEN (* Zeichen zu VALUE-String hinzufügen *)
    				pv := v_add; (* Zeichen eintragen *)
    				pv := pv + 1;
    				pv := 0; (* String-Terminierung eintragen *)
    			END_IF

    			i := i + 1; (* Datenzeiger erhöhen *)

    		END_IF
    	END_WHILE

    	CASE state OF
    	01:	(* Element gefunden *)
    		RESULT := 1; (* Element gefunden *)
    		OFFSET := i; (* OFFSET uebernehmen *)
    		RUN := 0;
    		state := 0;
    	02:	(* Element gefunden *)
    		RESULT := 2; (* Element und Zeilenende erkannt *)
    		OFFSET := i; (* OFFSET uebernehmen *)
    		RUN := 0;
    		state := 0;

    	05:	RESULT := 5; (* in Arbeit *)

    	10:	(* Indexüberschreitung - Bufferende *)
    		RESULT := 10; (* nichts gefunden - Datenende erreicht *)
    		OFFSET := i; (* OFFSET uebernehmen *)
    		RUN := 0;
    		state := 0;
    	END_CASE

    	(* ---------------- Debug-Message -----------------------*)
    	(*IF _debug_enable THEN
    		LOG_CL.NEW_MSG := 'CPF: intern RESULT ~1 , state ~2, step ~3 , OFFSET ~4, RUN ~5';
    		LOG_CL.PRINTF[1] := BYTE_TO_STRING(RESULT);
    		LOG_CL.PRINTF[2] := BYTE_TO_STRING(state);
    		LOG_CL.PRINTF[3] := INT_TO_STRING(step);
    		LOG_CL.PRINTF[4] := UDINT_TO_STRING(OFFSET);
    		LOG_CL.PRINTF[5] := BYTE_TO_STRING(RUN);
    		LOG_MSG();
    	END_IF*)
    	(* -----------------------------------------------------------------*)

    END_IF

    (* ---------------- Debug-Message -----------------------*)
    (*IF _debug_enable THEN
    	IF step_last <> step THEN
    		LOG_CL.NEW_MSG := 'IPB: step: ~1';
    		LOG_CL.PRINTF[1]  := INT_TO_STRING(step);
    		LOG_MSG();
    	END_IF
    	step_last := step;
    END_IF*)
    (* -----------------------------------------------------------------*)

    (* revision history
    ks	01. oct. 2010	rev 1.0
    	original version
    *)
END_FUNCTION_BLOCK

(* ---- CSV_PARSER_FILE.st ---- *)
FUNCTION_BLOCK CSV_PARSER_FILE
    (*http://www.oscat.de/images/OSCATNetwork/oscat_netlib121_en.pdf#page=149*)
    IF RUN > 0 THEN

    	IF state = 0 THEN (* Auswertung neu beginnen *)
    		pv := ADR(VALUE);
    		pv := 0; (* VALUE = '' *)
    		pve := pv + INT_TO_DWORD(STRING_LENGTH);
    		i := OFFSET;
    		RESULT := 0;
    		state := 5; (* Befehl in Arbeit (Busy) *)
    		step := 0; (* Auswertung neu beginnen *)

    		(* ---------------- Debug-Message -----------------------*)
    		(*IF _debug_enable THEN
    			LOG_CL.NEW_MSG := 'CPF: Startindex: ~1';
    			LOG_CL.PRINTF[1] := UDINT_TO_STRING(i);
    			LOG_MSG();
    		END_IF*)
    		(* -----------------------------------------------------------------*)

    	END_IF

    	watchdog(IN:=FALSE,PT:=T#1ms); (* Timer neustarten *)
    	watchdog.IN := TRUE;

    	WHILE (state = 5) DO (* Schleife solange kein Ergebnis *)

    		mode := 1;
    		FB(mode:=mode,FSD:=FSD,PT:=PT,FILENAME:=FILENAME,POS:=i );
    		e:=FB.ERROR;
    		c:=FB.DATA;

    		eof := i + 1 = FSD.FILE_SIZE; (* End of File *)

    		(* ---------------- Debug-Message -----------------------*)
    		(*IF _debug_enable THEN
    			LOG_CL.NEW_MSG := 'CPF: mode: ~1, error: ~2 , >~7<>~3< ~4 step ~5 index ~6';
    			LOG_CL.PRINTF[1] := BYTE_TO_STRING(mode);
    			LOG_CL.PRINTF[2] := BYTE_TO_STRING(e);
    			LOG_CL.PRINTF[3] := BYTE_TO_STRING(c);
    			LOG_CL.PRINTF[4] := BOOL_TO_STRING(eof);
    			LOG_CL.PRINTF[5] := INT_TO_STRING(step);
    			LOG_CL.PRINTF[6] := UDINT_TO_STRING(i);
    			LOG_CL.PRINTF[7] := CHR_TO_STRING(c);
    			LOG_MSG();
    		END_IF*)
    		(* -----------------------------------------------------------------*)
    		watchdog(); (* Timer aktualisieren *)

    		IF mode > 0 OR watchdog.Q THEN (* Baustein noch aktiv, oder watchdog ausgelöst *)
    			state := 5;
    			EXIT;
    		ELSIF e > 0 THEN (* File_error oder kein weiteres zeichen vorhanden *)
    			state := 10; (* nichts gefunden - Daten-Ende erreicht *)
    			EXIT;
    		ELSE

    			v_add := 0;

    			IF c = SEP THEN (* Neues Element erkannt *)
    				state := 1;
    				x := TRUE;
    			ELSIF c >= 32 THEN (* Element erkannt *)
    				v_add := c; (* Zeichen ablegen *)
    				IF eof THEN
    					state := 2; (* Element und Zeilenende erkannt *)
    				ELSE
    					x := TRUE;
    				END_IF
    			ELSE
    				IF x THEN
    					state := 2; (* Element und Zeilenende erkannt *)
    					x := FALSE;
    				END_IF
    			END_IF

    			IF v_add > 0  AND pv < pve THEN (* Zeichen zu VALUE-String hinzufügen *)
    				pv := v_add; (* Zeichen eintragen *)
    				pv := pv + 1;
    				pv := 0; (* String-Terminierung eintragen *)
    			END_IF

    			i := i + 1; (* Datenzeiger erhöhen *)

    		END_IF
    	END_WHILE

    	CASE state OF
    	01:	(* Element gefunden *)
    		RESULT := 1; (* Element gefunden *)
    		OFFSET := i; (* OFFSET uebernehmen *)
    		RUN := 0;
    		state := 0;
    	02:	(* Element gefunden *)
    		RESULT := 2; (* Element und Zeilenende erkannt *)
    		OFFSET := i; (* OFFSET uebernehmen *)
    		RUN := 0;
    		state := 0;

    	05:	RESULT := 5; (* in Arbeit *)

    	10:	(* Indexüberschreitung - Bufferende *)
    		RESULT := 10; (* nichts gefunden - Datenende erreicht *)
    		OFFSET := i; (* OFFSET uebernehmen *)
    		RUN := 0;
    		state := 0;
    	END_CASE

    	(* ---------------- Debug-Message -----------------------*)
    	(*IF _debug_enable THEN
    		LOG_CL.NEW_MSG := 'CPF: intern RESULT ~1 , state ~2, step ~3 , OFFSET ~4, RUN ~5';
    		LOG_CL.PRINTF[1] := BYTE_TO_STRING(RESULT);
    		LOG_CL.PRINTF[2] := BYTE_TO_STRING(state);
    		LOG_CL.PRINTF[3] := INT_TO_STRING(step);
    		LOG_CL.PRINTF[4] := UDINT_TO_STRING(OFFSET);
    		LOG_CL.PRINTF[5] := BYTE_TO_STRING(RUN);
    		LOG_MSG();
    	END_IF*)
    	(* -----------------------------------------------------------------*)

    END_IF

    (* ---------------- Debug-Message -----------------------*)
    (*IF _debug_enable THEN
    	IF step_last <> step THEN
    		LOG_CL.NEW_MSG := 'CPF: step: ~1';
    		LOG_CL.PRINTF[1]  := INT_TO_STRING(step);
    		LOG_MSG();
    	END_IF
    	step_last := step;
    END_IF*)
    (* -----------------------------------------------------------------*)

    (* revision history
    ks	01. oct. 2010	rev 1.0
    	original version
    *)
END_FUNCTION_BLOCK

(* ---- DLOG_BOOL.st ---- *)
FUNCTION_BLOCK DLOG_BOOL
    (*http://www.oscat.de/images/OSCATNetwork/oscat_netlib121_en.pdf#page=48*)
    CASE X.ADD_COM OF

    01:	(* ADD INFO *)
    	X.ID_MAX := X.ID_MAX + USINT#1;
    	id := WORD#16#0601; (* Quelltype BOOL , Zieltype STRING *)
    02:	(* ADD HEADER *)
    	X.UCB.D_STRING := COLUMN;
    	X.UCB.D_HEAD := id;
    	X.UCB.D_MODE := 1;
    	UCB(DATA:=X.UCB); (* Daten eintragen *)
    03:	(* ADD DATA *)
    	IF X.STORE_TYPE = BYTE#05 THEN (* MySQL-Modus *)
    		X.UCB.D_STRING := SEL(state_last,'0','1');
    	ELSE
    		X.UCB.D_STRING := SEL(state_last,OFF,ON);
    	END_IF
    	X.UCB.D_HEAD := id;

    	X.UCB.D_MODE := 1;
    	UCB(DATA:=X.UCB); (* Daten eintragen *)
    	last_delta := STATE;
    04:	(* ADD DATA REQ *)
    	IF DELTA AND (STATE XOR last_delta) THEN
    		X.ADD_DATA_REQ := TRUE;
    		last_delta := STATE;
    	END_IF
    END_CASE
    state_last := STATE;

    (* revision history
    ks	17. may. 2011	rev 1.0
    	original version

    ks	25. july.   2011	rev 1.1
    	neue head information

    ks	19. apr.   2012	rev 1.2
    	code neu überarbeitet

    *)
END_FUNCTION_BLOCK

(* ---- DLOG_CRON_TAB.st ---- *)
FUNCTION_BLOCK DLOG_CRON_TAB
    (*http://www.oscat.de/images/OSCATBasic/oscat_basic333_en.pdf#page=46*)
    IF ACTIVATE THEN
    	IF NOT activate_old THEN
    		CD.CE[0].VALUE_MIN := 0;	(* Sekunden *)
    		CD.CE[0].VALUE_MAX := 59;
    		CD.CE[1].VALUE_MIN := 0;	(* Minuten *)
    		CD.CE[1].VALUE_MAX := 59;
    		CD.CE[2].VALUE_MIN := 0;	(* Stunden *)
    		CD.CE[2].VALUE_MAX := 59;
    		CD.CE[3].VALUE_MIN := 1;	(* Tage *)
    		CD.CE[3].VALUE_MAX := 31;
    		CD.CE[4].VALUE_MIN := 1;	(* Wochentag *)
    		CD.CE[4].VALUE_MAX := 7;
    		CD.CE[5].VALUE_MIN := 1;	(* Monat *)
    		CD.CE[5].VALUE_MAX := 12;

    		FOR idx1 := 0 TO 5 DO
    			idx3 := CD.CE[idx1].VALUE_MIN;
    			idx4 := CD.CE[idx1].VALUE_MAx;
    			FOR idx2 := idx3 TO idx4 DO
    				CD.CE[idx1].ELEMENTS[idx2] := FALSE;
    			END_FOR
    			CD.CE[idx1].ALL_SELECTED := FALSE;
    		END_FOR

    		str1 := CONCAT(SECOND,'#');
    		str1 := CONCAT(str1,MINUTE);
    		str1 := CONCAT(str1,'#');
    		str1 := CONCAT(str1,HOUR);
    		str1 := CONCAT(str1,'#');
    		str1 := CONCAT(str1,DAY_OF_MONTH);
    		str1 := CONCAT(str1,'#');
    		str1 := CONCAT(str1,DAY_OF_WEEK);
    		str1 := CONCAT(str1,'#');
    		str1 := CONCAT(str1,MONTH);

    		FOR idx1 := 0 TO 5 DO
    			str2 := ELEMENT_GET(BYTE#35, idx1, str1);
    			IF LEN(str2) > 0 THEN
    				cnt1 := ELEMENT_COUNT(BYTE#44, str2);	(* Trenzeichen ',' *)
    			ELSE
    				cnt1 := 1;
    			END_IF

    			FOR idx2 := 0 TO cnt1 -1 DO
    				str3 := ELEMENT_GET(BYTE#44, idx2, str2);
    				IF FIND(str3, '*/') > 0 AND LEN(str3) <= 10 THEN
    					pos1 := DEC_TO_INT(str3);
    					IF pos1 > 0 THEN
    						idx3 := CD.CE[idx1].VALUE_MIN;
    						idx4 := CD.CE[idx1].VALUE_MAX;
    						WHILE idx3 <= idx4 DO
    							CD.CE[idx1].ELEMENTS[idx3] := TRUE;
    							idx3 := idx3 + pos1;
    						END_WHILE
    					END_IF

    				ELSE
    					IF FIND(str3, '*') > 0 OR LEN(str3) = 0 THEN
    						pos1 := CD.CE[idx1].VALUE_MIN;
    						pos2 := CD.CE[idx1].VALUE_MAX;
    						CD.CE[idx1].ALL_SELECTED := TRUE;
    					ELSE
    						cnt2 := ELEMENT_COUNT(BYTE#45, str3);	(* Trenzeichen '-' *)
    						char_cnt := LEN(str3);
    						IF char_cnt >= 1 AND char_cnt <= 10 THEN
    							num_str1 := ELEMENT_GET(BYTE#45, 0, str3);
    							pos1 := DEC_TO_INT(num_str1);
    							pos2 := pos1;
    							IF cnt2 = 2 THEN
    								num_str1 := ELEMENT_GET(BYTE#45, 1, str3);
    								pos2 := DEC_TO_INT(num_str1);
    							END_IF
    						END_IF
    					END_IF

    					IF pos1 >= CD.CE[idx1].VALUE_MIN AND pos2 <= CD.CE[idx1].VALUE_MAX THEN
    						FOR idx3 := pos1 TO pos2 DO
    							CD.CE[idx1].ELEMENTS[idx3] := TRUE;
    						END_FOR
    					END_IF
    				END_IF
    			END_FOR
    		END_FOR
    	ELSIF DTI <> dti_last THEN
    		CD.CE[0].VALUE := SECOND_OF_DT(DTI); (* Sekunden *)
    		CD.CE[1].VALUE := MINUTE_OF_DT(DTI); (* Minuten *)
    		CD.CE[2].VALUE := HOUR_OF_DT(DTI); (* Stunden *)
    		datei := DT_TO_DATE(DTI);
    		CD.CE[3].VALUE := DAY_OF_MONTH(datei); (* Tag *)
    		CD.CE[4].VALUE := DAY_OF_WEEK(datei); (* Wochentag *)
    		CD.CE[5].VALUE := MONTH_OF_DATE(datei); (*  Monat *)
    		dti_last := DTI;

    		idx2 := CD.CE[0].VALUE;	(* sekunden *)
    		Q := CD.CE[0].ELEMENTS[idx2] = TRUE;
    		idx2 := CD.CE[1].VALUE;	(* minuten *)
    		Q := Q AND CD.CE[1].ELEMENTS[idx2] = TRUE;
    		idx2 := CD.CE[2].VALUE;	(* stunden *)
    		Q := Q AND CD.CE[2].ELEMENTS[idx2] = TRUE;
    		idx2 := CD.CE[5].VALUE;	(* monat *)
    		Q := Q AND CD.CE[5].ELEMENTS[idx2] = TRUE;

    		(* auswertung Tag und Wochentag *)
    		idx2 := CD.CE[3].VALUE;	(* Tag *)
    		trig_day:= CD.CE[3].ELEMENTS[idx2] = TRUE;
    		idx2 := CD.CE[4].VALUE;	(* Wochentag *)
    		trig_weekday := CD.CE[4].ELEMENTS[idx2] = TRUE;

    		IF CD.CE[3].ALL_SELECTED = FALSE AND CD.CE[4].ALL_SELECTED = TRUE THEN
    			Q := Q AND trig_day; (* nur Tag auswerten *)
    		ELSIF CD.CE[3].ALL_SELECTED = TRUE AND CD.CE[4].ALL_SELECTED = FALSE THEN
    			Q := Q AND trig_weekday; (* nur Wochentag auswerten *)
    		ELSIF CD.CE[3].ALL_SELECTED = FALSE AND CD.CE[4].ALL_SELECTED = FALSE THEN
    			Q := Q AND (trig_weekday OR trig_day); (* Tag und Wochentag auswerten *)
    		END_IF
    	END_IF

    END_IF
    activate_old := ACTIVATE;

    (* revision history
    ks	27. oct. 2011	rev 1.0
    	original version
    *)
END_FUNCTION_BLOCK

(* ---- DLOG_DINT.st ---- *)
FUNCTION_BLOCK DLOG_DINT
    (*http://www.oscat.de/images/OSCATNetwork/oscat_netlib121_en.pdf#page=49*)
    CASE X.ADD_COM OF

    01:	(* ADD INFO *)
    	X.ID_MAX := X.ID_MAX + USINT#1;
    	id := WORD#16#0801; (* Quelltype DINT , Zieltype STRING *)
    02:	(* ADD HEADER *)
    	X.UCB.D_STRING := COLUMN;
    	X.UCB.D_HEAD := id;
    	X.UCB.D_MODE := 1;
    	UCB(DATA:=X.UCB); (* Daten eintragen *)
    03:	(* ADD DATA *)
    	X.UCB.D_STRING := DINT_TO_STRING(value_last);
    	X.UCB.D_HEAD := id;
    	X.UCB.D_MODE := 1;
    	UCB(DATA:=X.UCB); (* Daten eintragen *)
    	delta_last := value_last;
    04:	(* ADD DATA REQ *)
    	IF DELTA <> DINT#0 THEN
    		IF VALUE <= (delta_last - DELTA) OR VALUE >= (delta_last + DELTA) THEN
    			X.ADD_DATA_REQ := TRUE;
    			delta_last := VALUE;
    		END_IF
    	END_IF
    END_CASE
    value_last := VALUE;

    (* revision history
    ks	01. jan. 2011	rev 1.0
    	original version

    ks	17. may. 2011	rev 1.1
    	DELTA Funktion integriert

    ks	25. july.   2011	rev 1.2
    	neue head information

    ks	19. apr.   2012	rev 1.2
    	code neu überarbeitet
    *)
END_FUNCTION_BLOCK

(* ---- DLOG_DT.st ---- *)
FUNCTION_BLOCK DLOG_DT
    (*http://www.oscat.de/images/OSCATNetwork/oscat_netlib121_en.pdf#page=50*)
    CASE X.ADD_COM OF

    01:	(* ADD INFO *)
    	X.ID_MAX := X.ID_MAX + USINT#1;
    	id := WORD#16#0D01; (* Quelltype DT , Zieltype STRING *)
    02:	(* ADD HEADER *)
    	X.UCB.D_STRING := COLUMN;
    	X.UCB.D_HEAD := id;
    	X.UCB.D_MODE := 1;
    	UCB(DATA:=X.UCB); (* Daten eintragen *)
    03:	(* ADD DATA *)
    	X.UCB.D_STRING := DT_TO_STRF(DTI:=X.DTI,MS:=0,FMT:=FMT,LANG:=0);
    	X.UCB.D_HEAD := id;
    	X.UCB.D_MODE := 1;
    	UCB(DATA:=X.UCB); (* Daten eintragen *)
    	delta_last := X.DTI;
    04:	(* ADD DATA REQ *)
    	IF DELTA <> UDINT#0 THEN
    		IF DT_TO_UDINT(X.DTI) >= (DT_TO_UDINT(delta_last) + DELTA) THEN
    			X.ADD_DATA_REQ := TRUE;
    			delta_last := X.DTI;
    		END_IF
    	END_IF
    END_CASE

    (* revision history
    ks	01. jan. 2011	rev 1.0
    	original version

    ks	17. may. 2011	rev 1.1
    	COLUMN STRING(40), DELTA

    ks	25. july.   2011	rev 1.2
    	neue head information

    ks	19. apr.   2012	rev 1.3
    	code neu überarbeitet
    *)
END_FUNCTION_BLOCK

(* ---- DLOG_FILE_TO_FTP.st ---- *)
FUNCTION_BLOCK DLOG_FILE_TO_FTP
    (*http://www.oscat.de/images/OSCATNetwork/oscat_netlib121_en.pdf#page=63*)
    (* neue Filenamen speichern *)
    IF X.NEW_FILE_RTRIG AND ftrig_old = FALSE THEN
    	UCBD.D_HEAD := 1;
    	UCBD.D_MODE := 1;
    	UCBD.D_STRING := X.NEW_FILE;
    	UCB(DATA:=UCBD); (* Daten eintragen *)
    END_IF
    ftrig_old := X.NEW_FILE_RTRIG;

    CASE step OF

    00:	IF UCBD.BUF_COUNT > 0 AND ftp_busy = FALSE THEN
    		UCBD.D_MODE := 12; (* Daten lesen und löschen *)
    		UCB(DATA:=UCBD);
    		filename := UCBD.D_STRING;
    		cnt := RETRY;
    		step := 10;

    		(*####################  DEBUG-MESSAGE  ###################################*)
    		(*IF _debug_enable THEN
    			LOG_CL.NEW_MSG := 'F_T_FTP: Auftrag aktiv /file: ~2';
    			LOG_CL.PRINTF[2] := files;
    			LOG_MSG();
    		END_IF*)
    		(*########################################################################*)

    	END_IF

    10:	IF ftp_busy = FALSE THEN
    		IF ftp_done THEN
    			(*####################  DEBUG-MESSAGE  ###################################*)
    			(*IF _debug_enable THEN
    				LOG_CL.NEW_MSG := 'F_T_FTP: Auftrag OK /file: ~2';
    				LOG_CL.PRINTF[2] := filename;
    				LOG_MSG();
    			END_IF*)
    			(*########################################################################*)
    			step := 0;
    		ELSE
    			step := 20; (* pause nach error *)
    		END_IF
    	END_IF

    20:	IF WT_1.Q THEN (* Wartezeit *)
    		cnt := cnt - 1;
    		IF RETRY = 0 THEN (* FTP Transfer unbegrenzt wiederholen *)
    			(*####################  DEBUG-MESSAGE  ###################################*)
    			(*IF _debug_enable THEN
    				LOG_CL.NEW_MSG := 'F_T_FTP: Auftrag unbegrenzt wiederholen /file: ~2';
    				LOG_CL.PRINTF[2] := filename;
    				LOG_MSG();
    			END_IF*)
    			(*########################################################################*)
    			step := 10; (* FTP Transfer wiederholen *)
    		ELSIF cnt >= 0 THEN
    			(*####################  DEBUG-MESSAGE  ###################################*)
    			(*IF _debug_enable THEN
    				LOG_CL.NEW_MSG := 'F_T_FTP: Auftrag wiederholen /cnt: ~1 /file: ~2';
    				LOG_CL.PRINTF[1] := INT_TO_STRING(cnt);
    				LOG_CL.PRINTF[2] := filename;
    				LOG_MSG();
    			END_IF*)
    			(*########################################################################*)
    			step := 10; (* FTP Transfer wiederholen *)
    		ELSE
    			(*####################  DEBUG-MESSAGE  ###################################*)
    			(*IF _debug_enable THEN
    				LOG_CL.NEW_MSG := 'F_T_FTP: Auftrag verworfen /file: ~2';
    				LOG_CL.PRINTF[2] := filename;
    				LOG_MSG();
    			END_IF*)
    			(*########################################################################*)
    			step := 0; (* FTP Auftrag verwerfen *)
    		END_IF
    	END_IF

    END_CASE

    BUSY := step = 10;
    DONE := step = 0;
    WT_1(IN:= step = 20, PT:= RETRY_TIME);

    FTP_CLIENT(
    	ACTIVATE:= BUSY,
    	filename:= filename,
    	FTP_URL:= FTP_URL,
    	FTP_DOWNLOAD:= FALSE,
    	FTP_ACTIV:= FTP_ACTIV,
    	FILE_DELETE:= FILE_DELETE,
    	TIMEOUT:= TIMEOUT,
    	DNS_IP4:= DNS_IP4,
    	PLC_IP4:= PLC_IP4,
    	DONE=> ftp_done,
    	BUSY=> ftp_busy
    	);

    (* Fehlerauswertung *)
    IF FTP_CLIENT.ERROR_T <> BYTE#0 THEN
    	ERROR_C := FTP_CLIENT.ERROR_C;
    	ERROR_T := FTP_CLIENT.ERROR_T;
    ELSIF UCBD.BUF_DATA_LOST > UDINT#0 THEN
    	ERROR_C := DWORD#2; (* Fehler: Bufferüberlauf - Datenmenge reduzieren *)
    	ERROR_T := BYTE#6; 	(* Type: Buffer *)
    ELSIF UCBD.BUF_USED_MAX > USINT#90 THEN
    	ERROR_C := DWORD#1; (* Warnung: Buffer auslastung > 90% *)
    	ERROR_T := BYTE#6;	(* Type: Buffer *)
    ELSE
    	ERROR_C := DWORD#0;
    	ERROR_T := BYTE#0;
    END_IF

    (* revision history
    ks	01. jan. 2011	rev 1.0
    	original version

    ks	26. jul. 2011	rev 1.1
        codeoptimierung D_MODE 12

    ks	21. mar. 2016	rev 1.2
    	fehlermeldungen hinzugefügt
    	fehler in RETRY korrigiert

    *)
END_FUNCTION_BLOCK

(* ---- DLOG_FILE_TO_SMTP.st ---- *)
FUNCTION_BLOCK DLOG_FILE_TO_SMTP
    (*http://www.oscat.de/images/OSCATNetwork/oscat_netlib121_en.pdf#page=66*)
    (* neue Filenamen speichern *)
    IF X.NEW_FILE_RTRIG AND ftrig_old = FALSE THEN
    	UCBD.D_HEAD := 1;
    	UCBD.D_MODE := 1;
    	UCBD.D_STRING := X.NEW_FILE;
    	UCB(DATA:=UCBD); (* Daten eintragen *)
    END_IF
    ftrig_old := X.NEW_FILE_RTRIG;

    CASE step OF

    00:	IF UCBD.BUF_COUNT > 0 AND smtp_busy = FALSE THEN
    		UCBD.D_MODE := 12; (* Daten lesen und löschen *)
    		UCB(DATA:=UCBD);
    		files := UCBD.D_STRING;
    		IF FILE_DELETE THEN
    			files := CONCAT(files,';#DEL#');
    		END_IF
    		cnt := RETRY;
    		step := 10;

    		(*####################  DEBUG-MESSAGE  ###################################*)
    		(*IF _debug_enable THEN
    			LOG_CL.NEW_MSG := 'F_T_SMTP: Auftrag aktiv /file: ~2';
    			LOG_CL.PRINTF[2] := files;
    			LOG_MSG();
    		END_IF*)
    		(*########################################################################*)

    	END_IF

    10:	IF smtp_busy = FALSE THEN
    		IF smtp_done THEN
    			(*####################  DEBUG-MESSAGE  ###################################*)
    			(*IF _debug_enable THEN
    				LOG_CL.NEW_MSG := 'F_T_SMTP: Auftrag OK /file: ~2';
    				LOG_CL.PRINTF[2] := files;
    				LOG_MSG();
    			END_IF*)
    			(*########################################################################*)
    			step := 0;
    		ELSE
    			step := 20; (* pause nach error *)
    		END_IF
    	END_IF

    20:	IF WT_1.Q THEN (* Wartezeit *)
    		cnt := cnt - 1;
    		IF RETRY = 0 THEN (* Transfer unbegrenzt wiederholen *)
    			(*####################  DEBUG-MESSAGE  ###################################*)
    			(*IF _debug_enable THEN
    				LOG_CL.NEW_MSG := 'F_T_SMTP: Auftrag unbegrenzt wiederholen /file: ~2';
    				LOG_CL.PRINTF[2] := files;
    				LOG_MSG();
    			END_IF*)
    			(*########################################################################*)
    			step := 10; (* Transfer wiederholen *)
    		ELSIF cnt >= 0 THEN
    			(*####################  DEBUG-MESSAGE  ###################################*)
    			(*IF _debug_enable THEN
    				LOG_CL.NEW_MSG := 'F_T_SMTP: Auftrag wiederholen /cnt: ~1 /file: ~2';
    				LOG_CL.PRINTF[1] := INT_TO_STRING(cnt);
    				LOG_CL.PRINTF[2] := files;
    				LOG_MSG();
    			END_IF*)
    			(*########################################################################*)
    			step := 10; (* Transfer wiederholen *)
    		ELSE
    			(*####################  DEBUG-MESSAGE  ###################################*)
    			(*IF _debug_enable THEN
    				LOG_CL.NEW_MSG := 'F_T_SMTP: Auftrag verworfen /file: ~2';
    				LOG_CL.PRINTF[2] := files;
    				LOG_MSG();
    			END_IF*)
    			(*########################################################################*)
    			step := 0; (* Auftrag verwerfen *)
    		END_IF
    	END_IF

    END_CASE

    BUSY := step = 10;
    DONE := step = 0;
    WT_1(IN:= step = 20, PT:= RETRY_TIME);

    SMTP_CLIENT(
    	ACTIVATE:= BUSY,
    	TIMEOUT:= TIMEOUT,
    	DTI:= DTI,
    	DTI_OFFSET:= DTI_OFFSET,
    	DNS_IP4:= DNS_IP4,
    	SERVER:= SERVER,
    	MAILFROM:= MAILFROM,
    	MAILTO:= MAILTO,
    	SUBJECT:= SUBJECT,
    	BODY:= BODY,
    	files:= files,
    	DONE=> smtp_done,
    	BUSY=> smtp_busy
    	);

    (* Fehlerauswertung *)
    IF SMTP_CLIENT.ERROR_T <> BYTE#0 THEN
    	ERROR_C := SMTP_CLIENT.ERROR_C;
    	ERROR_T := SMTP_CLIENT.ERROR_T;
    ELSIF UCBD.BUF_DATA_LOST > UDINT#0 THEN
    	ERROR_C := DWORD#2; (* Fehler: Bufferüberlauf - Datenmenge reduzieren *)
    	ERROR_T := BYTE#6; 	(* Type: Buffer *)
    ELSIF UCBD.BUF_USED_MAX > USINT#90 THEN
    	ERROR_C := DWORD#1; (* Warnung: Buffer auslastung > 90% *)
    	ERROR_T := BYTE#6;	(* Type: Buffer *)
    ELSE
    	ERROR_C := DWORD#0;
    	ERROR_T := BYTE#0;
    END_IF

    (* revision history

    ks	01. jan. 2011	rev 1.0
    	original version

    ks	28. apr. 2011	rev 1.1
    	stringfehler bei option 'FILE_DELETE'

    ks	26. jul. 2011	rev 1.2
        codeoptimierung D_MODE 12

    ks	21. mar. 2016	rev 1.3
    	fehlermeldungen hinzugefügt
    	fehler in RETRY korrigiert

    *)
END_FUNCTION_BLOCK

(* ---- DLOG_REAL.st ---- *)
FUNCTION_BLOCK DLOG_REAL
    (*http://www.oscat.de/images/OSCATNetwork/oscat_netlib121_en.pdf#page=51*)
    CASE X.ADD_COM OF

    01:	(* ADD INFO *)
    	X.ID_MAX := X.ID_MAX + USINT#1;
    	id := WORD#16#0201; (* Quelltype REAL , Zieltype STRING *)
    02:	(* ADD HEADER *)
    	X.UCB.D_STRING := COLUMN;
    	X.UCB.D_HEAD := id;
    	X.UCB.D_MODE := 1;
    	UCB(DATA:=X.UCB); (* Daten eintragen *)
    03:	(* ADD DATA *)
    	X.UCB.D_STRING := REAL_TO_STRF(IN:=value_last,N:=N,D:=D);
    	X.UCB.D_HEAD := id;
    	X.UCB.D_MODE := 1;
    	UCB(DATA:=X.UCB); (* Daten eintragen *)
    	delta_last := value_last;
    04:	(* ADD DATA REQ *)
    	IF DELTA <> 0.0 THEN
    		IF VALUE <= (delta_last - DELTA) OR VALUE >= (delta_last + DELTA) THEN
    			X.ADD_DATA_REQ := TRUE;
    			delta_last := VALUE;
    		END_IF
    	END_IF
    END_CASE
    value_last := VALUE;

    (* revision history
    ks	01. jan. 2011	rev 1.0
    	original version

    ks	17. may. 2011	rev 1.1
    	DELTA Funktion integriert

    ks	25. july.   2011	rev 1.2
    	neue head information

    ks	19. apr.   2012	rev 1.3
    	code neu überarbeitet
    *)
END_FUNCTION_BLOCK

(* ---- DLOG_REAL_ARRAY.st ---- *)
FUNCTION_BLOCK DLOG_REAL_ARRAY
    (*http://www.oscat.de/images/OSCATBasic/oscat_basic333_en.pdf#page=46*)
    FOR idx := 1 TO R_COUNT DO

    	CASE X.ADD_COM OF

    	01:	(* ADD INFO *)
    		X.ID_MAX := X.ID_MAX + USINT#1;
    		id := WORD#16#0201; (* Quelltype REAL , Zieltype STRING *)
    		(* automatisch Namen vergeben *)
    		IF LEN(R_ARRAY[idx].COLUMN) = 0 THEN
    			R_ARRAY[idx].COLUMN := CONCAT('Spalte_',USINT_TO_STRING(X.ID_MAX));
    		END_IF
    	02:	(* ADD HEADER *)
    		X.UCB.D_STRING := R_ARRAY[idx].COLUMN;
    		X.UCB.D_HEAD := id;
    		X.UCB.D_MODE := 1;
    		UCB(DATA:=X.UCB); (* Daten eintragen *)
    	03:	(* ADD DATA *)
    		X.UCB.D_STRING := REAL_TO_STRF(IN:=R_ARRAY[idx]._value_last,N:=N,D:=D);
    		X.UCB.D_HEAD := id;
    		X.UCB.D_MODE := 1;
    		UCB(DATA:=X.UCB); (* Daten eintragen *)
    		R_ARRAY[idx]._delta_last := R_ARRAY[idx]._value_last;
    	04:	(* ADD DATA REQ *)
    		IF R_ARRAY[idx].DELTA <> 0.0 THEN
    			IF R_ARRAY[idx].VALUE <= (R_ARRAY[idx]._delta_last - R_ARRAY[idx].DELTA) OR R_ARRAY[idx].VALUE >= (R_ARRAY[idx]._delta_last + R_ARRAY[idx].DELTA) THEN
    				X.ADD_DATA_REQ := TRUE;
    				R_ARRAY[idx]._delta_last := R_ARRAY[idx].VALUE;
    			END_IF
    		END_IF
    	END_CASE
    	R_ARRAY[idx]._value_last := R_ARRAY[idx].VALUE;

    END_FOR

    (* revision history
    ks	03. mar. 2016	rev 1.0
    	original version

    *)
END_FUNCTION_BLOCK

(* ---- DLOG_STORE_FILE_CSV.st ---- *)
FUNCTION_BLOCK DLOG_STORE_FILE_CSV
    (*http://www.oscat.de/images/OSCATNetwork/oscat_netlib121_en.pdf#page=52*)
    X.DTI := DTI; (* Datum / Zeit eintragen *)
    X.CLOCK_TRIG := DTI <> dti_last;
    dti_last := DTI;
    trig_auto := FALSE;
    IF X.CLOCK_TRIG THEN (* Impuls in jeder Sekunde *)
    	fn := DT_TO_STRF(DTI, 0, FILENAME, 0); (* automatische Dateinamen generierung *)
    	IF TRIG_T >= T#1000ms THEN (* automatischer Trigger *)
    		trig_auto := DT_TO_UDINT(DTI) MOD (TIME_TO_UDINT(TRIG_T) / UDINT#1000) = UDINT#0;
    	END_IF
    END_IF

    CASE step_1 OF

    00:	IF ENABLE THEN
    		aw_enable := AUTO_CLOSE >= T#5s;
    		wd_time := SEL(X.LOAD_TIME_MAX > T#0s, T#5ms,X.LOAD_TIME_MAX);
    		fn_last := fn; (* aktuellen Dateinnamen speichern *)
    		IF X.ID_MAX = USINT#0 THEN (* nur einmal nach Satellitenbausteinen scannen *)
    			X.ADD_COM := 01; (* ADD INFO *)
    			X.STORE_TYPE := BYTE#2; (* CSV-Modus *)
    		END_IF
    		step_1 := 10;

    		(* ---------------- Debug-Message -----------------------*)
    		(*IF _debug_enable THEN
    			LOG_CL.NEW_MSG := 'FILE_CSV1 - Start: File [~1], [~2]';
    			LOG_CL.PRINTF[1] := fn_last;
    			LOG_CL.PRINTF[2] := DT_TO_STRING(DTI);
    			LOG_MSG();
    		END_IF*)
    		(* -----------------------------------------------------------------*)

    	END_IF

    10:	X.UCB.D_STRING := fn_last;
    	IF fn_last = SAVE_DATA.FN_REM THEN
    		X.UCB.D_HEAD := WORD#16#F201; (* Filemode open + write *)
    		X.ADD_COM := 00;
    	ELSE
    		X.UCB.D_HEAD := WORD#16#F301; (* Filemode create + write *)
    		X.ADD_COM := 02; (* ADD HEADER *)
    	END_IF

    	X.UCB.D_MODE := 1; (* Dateinamen als String ablegen *)
    	UCB(DATA:=X.UCB); (* Daten eintragen *)
    	step_1 := 30;

    30:	(* LOG-Trigger verarbeiten *)
    	trig_tmp := (TRIG_M AND NOT trig_m_last) OR trig_auto OR X.ADD_DATA_REQ;

    	IF ENABLE = FALSE OR fn <> fn_last THEN (* ENABLE = 0 oder neuen Dateinamen -> Log Stop *)
    		trig_stored := trig_tmp; (* aktuellen Triggerpuls speichern *)
    		X.UCB.D_HEAD := WORD#16#EE00;
    		X.UCB.D_MODE := 1;
    		UCB(DATA:=X.UCB); (* Element schreiben *)
    		X.ADD_COM := 00;
    		step_1 := 00;

    		(* ---------------- Debug-Message -----------------------*)
    		(*IF _debug_enable THEN
    			LOG_CL.NEW_MSG := 'FILE_CSV1 - Stop: [~2]';
    			LOG_CL.PRINTF[2] := DT_TO_STRING(DTI);
    			LOG_MSG();
    		END_IF*)
    		(* -----------------------------------------------------------------*)

    	ELSIF ENABLE THEN
    		IF trig_tmp OR trig_stored THEN (* manueller, automatischer oder externer Trigger *)
    			trig_stored := FALSE;
    			X.ADD_COM := 03; (* ADD DATA *)
    			SAVE_DATA.TRIG_CNT := SAVE_DATA.TRIG_CNT + UDINT#1;
    			SAVE_DATA.TRIG_CNT_TOTAL  := SAVE_DATA.TRIG_CNT_TOTAL + UDINT#1;
    			(* ---------------- Debug-Message -----------------------*)
    			(*IF _debug_enable THEN
    				LOG_CL.NEW_MSG := 'FILE_CSV1 - Trig: [~2]';
    				LOG_CL.PRINTF[2] := DT_TO_STRING(DTI);
    				LOG_MSG();
    			END_IF*)
    			(* -----------------------------------------------------------------*)
    		ELSE
    			X.ADD_COM := 04;	(* ADD DATA REQ *)
    		END_IF
    	END_IF

    END_CASE
    X.ADD_DATA_REQ := FALSE; (* externe Anforderung rücksetzen *)

    (* ##################################### *)

    CASE step_2 OF

    00:	aw_ton(IN:= idx > 0 AND aw_enable, PT:= AUTO_CLOSE); (* AutoWrite Timer *)
    	IF aw_ton.Q THEN (* Zeitgesteuertes Datenschreiben *)
    		aw_aktiv := TRUE;
    		step_2 := 10; (* Daten schreiben *)
    		(* ---------------- Debug-Message -----------------------*)
    		(*IF _debug_enable THEN
    			LOG_CL.NEW_MSG := 'FILE_CSV2 - AutoWrite: [~2]';
    			LOG_CL.PRINTF[2] := DT_TO_STRING(DTI);
    			LOG_MSG();
    		END_IF*)
    		(* -----------------------------------------------------------------*)

    	ELSE
    		wd_ton(IN:= FALSE, PT:= wd_time);
    		wd_ton(IN:= TRUE);
    		WHILE X.UCB.BUF_COUNT > 0 AND step_2 = 0 AND wd_ton.Q = FALSE DO

    			X.UCB.D_MODE := 10;
    			UCB(DATA:=X.UCB); (* Element lesen , aber noch nicht entfernen *)
    			IF X.UCB.D_HEAD > WORD#16#F000 THEN (* F301 oder F201 *)
    				X.UCB.D_MODE := 11;
    				UCB(DATA:=X.UCB); (* Element entfernen *)

    				FSD.MODE := WORD_TO_BYTE(SHR(SHL(X.UCB.D_HEAD,4),12)); (* 0X00 -> 000X = 3 create + write / 2 open + write *)
    				FSD.OFFSET := UDINT#0; (* Start bei Dateianfang *)
    				FSD.FILENAME := X.UCB.D_STRING; (* Dateiname *)
    				PT.SIZE := UINT#0;
    				SAVE_DATA.FN_REM := FSD.FILENAME; (* aktuellen Dateinamen remanent sichern *)

    				IF FSD.MODE = BYTE#3 THEN	(* Datei neu anlegen -> dann zähler reset *)
    					SAVE_DATA.TRIG_CNT := UDINT#0;
    				END_IF

    				X.NEW_FILE := FSD.FILENAME;
    				X.NEW_FILE_SIZE := UDINT#0;
    				X.NEW_FILE_RTRIG := FALSE;
    				step_2 := 20;
    				(* ---------------- Debug-Message -----------------------*)
    				(*IF _debug_enable THEN
    					LOG_CL.NEW_MSG := 'FILE_CSV2 - Create: Mode [~1] , [~2]';
    					LOG_CL.PRINTF[2] := DT_TO_STRING(DTI);
    					LOG_CL.PRINTF[1] := BYTE_TO_STRING(FSD.MODE);
    					LOG_MSG();
    				END_IF*)
    				(* -----------------------------------------------------------------*)

    			ELSIF X.UCB.D_HEAD = WORD#16#EE00 THEN (* log_stop Command *)
    				X.UCB.D_MODE := 11;
    				UCB(DATA:=X.UCB); (* Element entfernen *)
    				log_stop := TRUE;
    				step_2 := 10; (* Daten schreiben *)

    			ELSIF idx + X.UCB.D_SIZE + 2 < SIZEOF(PT.BUFFER) THEN (* bufferplatz vorhanden *)
    				X.UCB.D_MODE := 11;
    				UCB(DATA:=X.UCB); (* Element entfernen *)
    				(* ---------------- Debug-Message -----------------------*)
    				(*IF _debug_enable THEN
    					LOG_CL.NEW_MSG := 'FILE_CSV2 - BUF: TXT [~1],Pos [~2], [~3]';
    					LOG_CL.PRINTF[1] := X.UCB.D_STRING;
    					LOG_CL.PRINTF[2] := INT_TO_STRING(idx);
    					LOG_CL.PRINTF[3] := DT_TO_STRING(DTI);
    					LOG_MSG();
    				END_IF*)
    				(* -----------------------------------------------------------------*)
    				_STRING_TO_BUFFER(STR:=X.UCB.D_STRING, POS:=idx, PT:=ADR(PT.BUFFER), SIZE:=SIZEOF(PT.BUFFER));
    				idx := idx + LEN(X.UCB.D_STRING);
    				n := n + USINT#1;
    				IF n = X.ID_MAX THEN (* letztes Element einer Zeile *)
    					n := USINT#0;
    					PT.BUFFER[idx] := BYTE#16#0D;
    					idx := idx + 1;
    					PT.BUFFER[idx] := BYTE#16#0A;
    				ELSE
    					PT.BUFFER[idx] := SEP;
    				END_IF
    				idx := idx + 1;
    				X.NEW_FILE_SIZE := total_bytes + INT_TO_UDINT(idx);
    			ELSE (* kein Platz vorhanden *)
    				step_2 := 10; (* Daten schreiben *)
    			END_IF
    			wd_ton();
    		END_WHILE
    	END_IF

    10:	IF idx > 0 THEN (* Daten schreiben *)
    		FSD.MODE := BYTE#2; (* File_Open_Exist + File_Write *)
    		FSD.OFFSET := UDINT#4294967294; (* 16#FFFF_FFFE ->Spezialcode: Daten automatisch an Dateiende anhängen *)
    		PT.SIZE := INT_TO_UINT(idx); (* Datenlänge eintragen *)
    		idx := 0;
    		(* ---------------- Debug-Message -----------------------*)
    		(*IF _debug_enable THEN
    			LOG_CL.NEW_MSG := 'FILE_CSV2 - WriteData: Mode [~3] Size [~1] , [~2]';
    			LOG_CL.PRINTF[1] := UINT_TO_STRING(PT.SIZE);
    			LOG_CL.PRINTF[2] := DT_TO_STRING(DTI);
    			LOG_CL.PRINTF[3] := BYTE_TO_STRING(FSD.MODE);
    			LOG_MSG();
    		END_IF*)
    		(* -----------------------------------------------------------------*)
    	END_IF
    	step_2 := 20;

    20:	IF FSD.MODE = BYTE#0 THEN
    		total_bytes := FSD.FILE_SIZE;
    		X.NEW_FILE_SIZE := total_bytes + INT_TO_UDINT(idx);
    		IF log_stop OR aw_aktiv THEN
    			aw_aktiv := FALSE;
    			FSD.MODE := BYTE#5; (* Datei schliessen *)
    			(* ---------------- Debug-Message -----------------------*)
    			(*IF _debug_enable THEN
    				LOG_CL.NEW_MSG := 'FILE_CSV2 - Close: [~2]';
    				LOG_CL.PRINTF[2] := DT_TO_STRING(DTI);
    				LOG_MSG();
    			END_IF*)
    			(* -----------------------------------------------------------------*)
    		END_IF
    		step_2 := 30;
    	END_IF

    30:	IF FSD.MODE = BYTE#0 THEN (* Befehl beendet ? *)
    		IF log_stop THEN
    			X.NEW_FILE_RTRIG := TRUE;
    			log_stop := FALSE;
    			SAVE_DATA.FN_REM := ''; (* remanenten Dateinamen löschen *)
    		END_IF
    		step_2 := 00;
    	END_IF

    END_CASE

    FS(FSD:=FSD,PT:=PT); (* FILE_SERVER *)
    (* Fehlerauswertung *)
    IF FSD.ERROR <> BYTE#0 THEN
    	ERROR_C := BYTE_TO_DWORD(FSD.ERROR);
    	ERROR_T := BYTE#1;
    ELSIF X.UCB.BUF_DATA_LOST > UDINT#0 THEN
    	ERROR_C := DWORD#2; (* Fehler: Bufferüberlauf - Datenmenge reduzieren *)
    	ERROR_T := BYTE#6; 	(* Type: Buffer *)
    ELSIF X.UCB.BUF_USED_MAX > USINT#90 THEN
    	ERROR_C := DWORD#1; (* Warnung: Buffer auslastung > 90% *)
    	ERROR_T := BYTE#6;	(* Type: Buffer *)
    ELSE
    	ERROR_C := DWORD#0;
    	ERROR_T := BYTE#0;
    END_IF

    trig_m_last := TRIG_M;

    (* revision history
    ks	01. jan. 2011	rev 1.0
    	original version

    ks	13. may. 2011	rev 1.1
    	ADD_DATA_REQ, ERROR_T, ERROR_C hinzugefügt

    ks	25. july. 2011	rev 1.2
    	HEAD Informationen geändert, neuer Spaltenzähler

    ks	16. apr. 2012	rev 1.3
    	neuer überarbeiteter Code für automatisches File-open/close

    ks	8. mar. 2016	rev 1.4
    	nur einmal nach satellitenbausteinen scannen

    ks	21. mar. 2016	rev 1.5
    	prüfung auf freien bufferplatz hinzugefügt
    	fehlermeldungen hinzugefügt
    *)
END_FUNCTION_BLOCK

(* ---- DLOG_STORE_FILE_HTML.st ---- *)
FUNCTION_BLOCK DLOG_STORE_FILE_HTML
    (*http://www.oscat.de/images/OSCATBasic/oscat_basic333_en.pdf#page=46*)
    X.DTI := DTI; (* Datum / Zeit eintragen *)
    X.CLOCK_TRIG := DTI <> dti_last;
    dti_last := DTI;
    trig_auto := FALSE;
    IF X.CLOCK_TRIG THEN (* Impuls in jeder Sekunde *)
    	fn := DT_TO_STRF(DTI, 0, FILENAME, 0); (* automatische Dateinamen generierung *)
    	IF TRIG_T >= T#1000ms THEN (* automatischer Trigger *)
    		trig_auto := DT_TO_UDINT(DTI) MOD (TIME_TO_UDINT(TRIG_T) / UDINT#1000) = UDINT#0;
    	END_IF
    END_IF

    CASE step_1 OF

    00:	IF ENABLE THEN
    		aw_enable := AUTO_CLOSE >= T#5s;
    		wd_time := SEL(X.LOAD_TIME_MAX > T#0s, T#5ms,X.LOAD_TIME_MAX);
    		fn_last := fn; (* aktuellen Dateinnamen speichern *)
    		IF X.ID_MAX = USINT#0 THEN (* nur einmal nach Satellitenbausteinen scannen *)
    			X.ADD_COM := 01; (* ADD INFO *)
    			X.STORE_TYPE := BYTE#4; (* HTML-Modus *)
    		END_IF
    		step_1 := 10;

    		(* ---------------- Debug-Message -----------------------*)
    		(*IF _debug_enable THEN
    			LOG_CL.NEW_MSG := 'FILE_HTML1 - Start: File [~1], [~2]';
    			LOG_CL.PRINTF[1] := fn_last;
    			LOG_CL.PRINTF[2] := DT_TO_STRING(DTI);
    			LOG_MSG();
    		END_IF*)
    		(* -----------------------------------------------------------------*)

    	END_IF

    10:	X.UCB.D_STRING := fn_last;
    	IF fn_last = SAVE_DATA.FN_REM THEN
    		X.UCB.D_HEAD := WORD#16#F201; (* Filemode open + write *)
    		X.ADD_COM := 00;
    	ELSE
    		X.UCB.D_HEAD := WORD#16#F301; (* Filemode create + write *)
    		X.ADD_COM := 02; (* ADD HEADER *)
    	END_IF

    	X.UCB.D_MODE := 1; (* Dateinamen als String ablegen *)
    	UCB(DATA:=X.UCB); (* Daten eintragen *)
    	step_1 := 30;

    30:	(* LOG-Trigger verarbeiten *)
    	trig_tmp := (TRIG_M AND NOT trig_m_last) OR trig_auto OR X.ADD_DATA_REQ;

    	IF ENABLE = FALSE OR fn <> fn_last THEN (* ENABLE = 0 oder neuen Dateinamen -> Log Stop *)
    		trig_stored := trig_tmp; (* aktuellen Triggerpuls speichern *)
    		X.UCB.D_HEAD := WORD#16#EE00;
    		X.UCB.D_MODE := 1;
    		UCB(DATA:=X.UCB); (* Element schreiben *)
    		X.ADD_COM := 00;
    		step_1 := 00;

    		(* ---------------- Debug-Message -----------------------*)
    		(*IF _debug_enable THEN
    			LOG_CL.NEW_MSG := 'FILE_HTML1 - Stop: [~2]';
    			LOG_CL.PRINTF[2] := DT_TO_STRING(DTI);
    			LOG_MSG();
    		END_IF*)
    		(* -----------------------------------------------------------------*)

    	ELSIF ENABLE THEN
    		IF trig_tmp OR trig_stored THEN (* manueller, automatischer oder externer Trigger *)
    			trig_stored := FALSE;
    			X.ADD_COM := 03; (* ADD DATA *)
    			SAVE_DATA.TRIG_CNT := SAVE_DATA.TRIG_CNT + UDINT#1;
    			SAVE_DATA.TRIG_CNT_TOTAL  := SAVE_DATA.TRIG_CNT_TOTAL + UDINT#1;
    			(* ---------------- Debug-Message -----------------------*)
    			(*IF _debug_enable THEN
    				LOG_CL.NEW_MSG := 'FILE_HTML1 - Trig: [~2]';
    				LOG_CL.PRINTF[2] := DT_TO_STRING(DTI);
    				LOG_MSG();
    			END_IF*)
    			(* -----------------------------------------------------------------*)
    		ELSE
    			X.ADD_COM := 04;	(* ADD DATA REQ *)
    		END_IF
    	END_IF

    END_CASE
    X.ADD_DATA_REQ := FALSE; (* externe Anforderung rücksetzen *)

    (* ##################################### *)

    CASE step_2 OF

    00:	aw_ton(IN:= idx > 0 AND aw_enable , PT:= AUTO_CLOSE); (* AutoWrite Timer *)
    	IF aw_ton.Q THEN (* Zeitgesteuertes Datenschreiben *)
    		aw_aktiv := TRUE;
    		step_2 := 10; (* Daten schreiben *)
    		(* ---------------- Debug-Message -----------------------*)
    		(*IF _debug_enable THEN
    			LOG_CL.NEW_MSG := 'FILE_HTML2 - AutoWrite: [~2]';
    			LOG_CL.PRINTF[2] := DT_TO_STRING(DTI);
    			LOG_MSG();
    		END_IF*)
    		(* -----------------------------------------------------------------*)

    	ELSE
    		wd_ton(IN:= FALSE, PT:= wd_time);
    		wd_ton(IN:= TRUE);
    		WHILE X.UCB.BUF_COUNT > 0 AND step_2 = 0 AND wd_ton.Q = FALSE DO

    			X.UCB.D_MODE := 10;
    			UCB(DATA:=X.UCB); (* Element lesen , aber noch nicht entfernen *)

    			IF X.UCB.D_HEAD > WORD#16#F000 THEN (* F301 oder F201 *)

    				str := CONCAT('<html><body><table ',HTML_TABLE);
    		        		str := CONCAT(str,'><caption>');
    		        		str := CONCAT(str,HTML_CAPTION);
    		        		str := CONCAT(str,'</caption>');

    				IF idx + LEN(str) < SIZEOF(PT.BUFFER) THEN (* Platz für Element vorhanden ? *)

    					FSD.MODE := WORD_TO_BYTE(SHR(SHL(X.UCB.D_HEAD,4),12)); (* 0X00 -> 000X = 3 create + write / 2 open + write *)
    					FSD.OFFSET := UDINT#0; (* Start bei Dateianfang *)
    					FSD.FILENAME := X.UCB.D_STRING; (* Dateiname *)
    					PT.SIZE := UINT#0;
    					SAVE_DATA.FN_REM := FSD.FILENAME; (* aktuellen Dateinamen remanent sichern *)

    					X.NEW_FILE := FSD.FILENAME;
    					X.NEW_FILE_SIZE := UDINT#0;
    					X.NEW_FILE_RTRIG := FALSE;
    					step_2 := 20;

    					(* Headerdaten schreiben *)
    					IF FSD.MODE = BYTE#3 THEN
    						SAVE_DATA.TRIG_CNT := UDINT#0; (* Datei neu anlegen -> dann zähler reset *)
    						SAVE_DATA.COLOR := FALSE;
    						SAVE_DATA.HEAD := FALSE;

    						_STRING_TO_BUFFER(str:=str, POS:=idx, PT:=ADR(PT.BUFFER), SIZE:=SIZEOF(PT.BUFFER));
    						idx := idx + LEN(str);
    						X.NEW_FILE_SIZE := total_bytes + INT_TO_UDINT(idx);
    					END_IF

    					X.UCB.D_MODE := 11;
    					UCB(DATA:=X.UCB); (* Element entfernen *)

    					(* ---------------- Debug-Message -----------------------*)
    					(*IF _debug_enable THEN
    						LOG_CL.NEW_MSG := 'FILE_HTML2 - Create: Mode [~1] , [~2]';
    						LOG_CL.PRINTF[2] := DT_TO_STRING(DTI);
    						LOG_CL.PRINTF[1] := BYTE_TO_STRING(FSD.MODE);
    						LOG_MSG();
    					END_IF*)
    					(* -----------------------------------------------------------------*)
    				END_IF

    			ELSIF X.UCB.D_HEAD = WORD#16#EE00 THEN (* log_stop Command *)

    				str := '</table></body></html>';

    				IF idx + LEN(str) < SIZEOF(PT.BUFFER) THEN (* Platz für Element vorhanden ? *)

    					_STRING_TO_BUFFER(str:=str, POS:=idx, PT:=ADR(PT.BUFFER), SIZE:=SIZEOF(PT.BUFFER));
    					idx := idx + LEN(str);
    					log_stop := TRUE;
    					step_2 := 10; (* Daten schreiben *)

    					X.UCB.D_MODE := 11;
    					UCB(DATA:=X.UCB); (* Element entfernen *)
    				END_IF

    			ELSIF idx + LEN(X.UCB.D_STRING) + 120 < SIZEOF(PT.BUFFER) THEN (* Platz für Element vorhanden ? *)

    				(* ---------------- Debug-Message -----------------------*)
    				(*IF _debug_enable THEN
    					LOG_CL.NEW_MSG := 'FILE_CSV2 - BUF: TXT [~1],Pos [~2], [~3]';
    					LOG_CL.PRINTF[1] := X.UCB.D_STRING;
    					LOG_CL.PRINTF[2] := INT_TO_STRING(idx);
    					LOG_CL.PRINTF[3] := DT_TO_STRING(DTI);
    					LOG_MSG();
    				END_IF*)
    				(* -----------------------------------------------------------------*)

    				IF log_state = USINT#0 THEN
    					str := '<TR ';
    					IF NOT SAVE_DATA.HEAD THEN
    						str := CONCAT(str,HTML_TR_HEAD);
    						SAVE_DATA.HEAD := TRUE;
    					ELSIF SAVE_DATA.COLOR THEN
    						str := CONCAT(str,HTML_TR_EVEN);
    					ELSE
    						str := CONCAT(str,HTML_TR_ODD);
    					END_IF
    					str := CONCAT(str,'><TD>');
    				ELSE
    					str := '<TD>';
    				END_IF

    				_STRING_TO_BUFFER(str:=str, POS:=idx, PT:=ADR(PT.BUFFER), SIZE:=SIZEOF(PT.BUFFER));
    				idx := idx + LEN(str);
    				log_state := log_state + USINT#1;

    				_STRING_TO_BUFFER(str:=X.UCB.D_STRING, POS:=idx, PT:=ADR(PT.BUFFER), SIZE:=SIZEOF(PT.BUFFER));
    				idx := idx + LEN(X.UCB.D_STRING);
    				n := n + USINT#1;
    				IF n >= X.ID_MAX THEN
    					n := USINT#0;
    					str := '</TD></TR>';
    					SAVE_DATA.COLOR := NOT SAVE_DATA.COLOR;
    					log_state := USINT#0;
    				ELSE
    					str := '</TD>';
    				END_IF
    				_STRING_TO_BUFFER(str:=str, POS:=idx, PT:=ADR(PT.BUFFER), SIZE:=SIZEOF(PT.BUFFER));
    				idx := idx + LEN(str);
    				X.NEW_FILE_SIZE := total_bytes + INT_TO_UDINT(idx);

    				X.UCB.D_MODE := 11;
    				UCB(DATA:=X.UCB); (* Element entfernen *)

    			ELSE (* kein Platz vorhanden *)
    				step_2 := 10; (* Daten schreiben *)

    			END_IF
    			wd_ton();
    		END_WHILE
    	END_IF

    10:	IF idx > 0 THEN (* Daten schreiben *)
    		FSD.MODE := BYTE#2; (* File_Open_Exist + File_Write *)
    		FSD.OFFSET := UDINT#4294967294; (* 16#FFFF_FFFE ->Spezialcode: Daten automatisch an Dateiende anhängen *)
    		PT.SIZE := INT_TO_UINT(idx); (* Datenlänge eintragen *)
    		idx := 0;
    		(* ---------------- Debug-Message -----------------------*)
    		(*IF _debug_enable THEN
    			LOG_CL.NEW_MSG := 'FILE_HTML2 - WriteData: Mode [~3] Size [~1] , [~2]';
    			LOG_CL.PRINTF[1] := UINT_TO_STRING(PT.SIZE);
    			LOG_CL.PRINTF[2] := DT_TO_STRING(DTI);
    			LOG_CL.PRINTF[3] := BYTE_TO_STRING(FSD.MODE);
    			LOG_MSG();
    		END_IF*)
    		(* -----------------------------------------------------------------*)
    	END_IF
    	step_2 := 20;

    20:	IF FSD.MODE = BYTE#0 THEN
    		total_bytes := FSD.FILE_SIZE;
    		X.NEW_FILE_SIZE := total_bytes + INT_TO_UDINT(idx);
    		IF log_stop OR aw_aktiv THEN
    			aw_aktiv := FALSE;
    			FSD.MODE := BYTE#5; (* Datei schliessen *)
    			(* ---------------- Debug-Message -----------------------*)
    			(*IF _debug_enable THEN
    				LOG_CL.NEW_MSG := 'FILE_HTML2 - Close: [~2]';
    				LOG_CL.PRINTF[2] := DT_TO_STRING(DTI);
    				LOG_MSG();
    			END_IF*)
    			(* -----------------------------------------------------------------*)
    		END_IF
    		step_2 := 30;
    	END_IF

    30:	IF FSD.MODE = BYTE#0 THEN (* Datei schliessen beendet *)
    		IF log_stop THEN
    			X.NEW_FILE_RTRIG := TRUE;
    			log_stop := FALSE;
    			SAVE_DATA.FN_REM := ''; (* remanenten Dateinamen löschen *)
    		END_IF
    		step_2 := 00;
    	END_IF

    END_CASE

    FS(FSD:=FSD,PT:=PT); (* FILE_SERVER *)

    (* Fehlerauswertung *)
    IF FSD.ERROR <> BYTE#0 THEN
    	ERROR_C := BYTE_TO_DWORD(FSD.ERROR);
    	ERROR_T := BYTE#1;
    ELSIF X.UCB.BUF_DATA_LOST > UDINT#0 THEN
    	ERROR_C := DWORD#2; (* Fehler: Bufferüberlauf - Datenmenge reduzieren *)
    	ERROR_T := BYTE#6; 	(* Type: Buffer *)
    ELSIF X.UCB.BUF_USED_MAX > USINT#90 THEN
    	ERROR_C := DWORD#1; (* Warnung: Buffer auslastung > 90% *)
    	ERROR_T := BYTE#6;	(* Type: Buffer *)
    ELSE
    	ERROR_C := DWORD#0;
    	ERROR_T := BYTE#0;
    END_IF

    trig_m_last := TRIG_M;

    (* revision history
    ks	25. july. 2011	rev 1.0
    	original version

    ks	16. apr. 2012	rev 1.1
    	neuer überarbeiteter Code für automatisches File-open/close

    ks	8. mar. 2016	rev 1.2
    	nur einmal nach satellitenbausteinen scannen

    ks	21. mar. 2016	rev 1.3
    	prüfung auf freien bufferplatz hinzugefügt
    	fehlermeldungen hinzugefügt

    *)
END_FUNCTION_BLOCK
